LIN {X 0.037,Y -515.295,Z 622.606,A 0.000,B 0.000,C 90.000,E1 325.022} C_DIS
LIN {X 0.251,Y -517.921,Z 622.601,A 0.000,B 0.000,C 90.000,E1 324.116} C_DIS
LIN {X 0.091,Y -520.064,Z 622.598,A 0.000,B 0.000,C 90.000,E1 323.623} C_DIS
LIN {X 0.035,Y -521.634,Z 622.596,A 0.000,B 0.000,C 90.000,E1 323.336} C_DIS
LIN {X 0.167,Y -524.111,Z 622.594,A 0.000,B 0.000,C 90.000,E1 322.924} C_DIS
LIN {X 0.183,Y -527.814,Z 622.592,A 0.000,B 0.000,C 90.000,E1 322.477} C_DIS
LIN {X 0.246,Y -531.406,Z 622.590,A 0.000,B 0.000,C 90.000,E1 322.110} C_DIS
LIN {X -0.214,Y -538.842,Z 622.586,A 0.000,B 0.000,C 90.000,E1 321.537} C_DIS
LIN {X -0.001,Y -548.855,Z 622.582,A 0.000,B 0.000,C 90.000,E1 320.723} C_DIS
LIN {X -0.006,Y -561.804,Z 622.576,A 0.000,B 0.000,C 90.000,E1 319.666} C_DIS
LIN {X -0.280,Y -573.310,Z 622.571,A 0.000,B 0.000,C 90.000,E1 318.771} C_DIS
LIN {X 0.089,Y -581.806,Z 622.567,A 0.000,B 0.000,C 90.000,E1 318.038} C_DIS
LIN {X -0.035,Y -595.533,Z 622.560,A 0.000,B 0.000,C 90.000,E1 316.863} C_DIS
LIN {X 0.149,Y -600.581,Z 622.558,A 0.000,B 0.000,C 90.000,E1 316.377} C_DIS
LIN {X -0.381,Y -605.341,Z 622.555,A 0.000,B 0.000,C 90.000,E1 315.972} C_DIS
LIN {X 0.005,Y -609.117,Z 622.553,A 0.000,B 0.000,C 90.000,E1 315.567} C_DIS
LIN {X 0.270,Y -612.804,Z 622.551,A 0.000,B 0.000,C 90.000,E1 315.162} C_DIS
LIN {X 0.162,Y -620.880,Z 622.546,A 0.000,B 0.000,C 90.000,E1 314.271} C_DIS
LIN {X 0.244,Y -626.155,Z 622.543,A 0.000,B 0.000,C 90.000,E1 313.623} C_DIS
LIN {X -0.183,Y -633.203,Z 622.538,A 0.000,B 0.000,C 90.000,E1 312.771} C_DIS
LIN {X -0.232,Y -643.744,Z 622.530,A 0.000,B 0.000,C 90.000,E1 311.391} C_DIS
LIN {X 0.027,Y -650.113,Z 622.525,A 0.000,B 0.000,C 90.000,E1 310.496} C_DIS
LIN {X -0.084,Y -654.219,Z 622.522,A 0.000,B 0.000,C 90.000,E1 309.886} C_DIS
LIN {X -0.165,Y -657.973,Z 622.518,A 0.000,B 0.000,C 90.000,E1 309.277} C_DIS
LIN {X 0.262,Y -660.763,Z 622.515,A 0.000,B 0.000,C 90.000,E1 308.749} C_DIS
LIN {X -0.223,Y -663.342,Z 622.513,A 0.000,B 0.000,C 90.000,E1 308.302} C_DIS
LIN {X 0.327,Y -666.913,Z 622.509,A 0.000,B 0.000,C 90.000,E1 307.523} C_DIS
LIN {X -0.018,Y -670.263,Z 622.505,A 0.000,B 0.000,C 90.000,E1 306.824} C_DIS
LIN {X -0.058,Y -672.250,Z 622.502,A 0.000,B 0.000,C 90.000,E1 306.343} C_DIS
LIN {X 0.053,Y -674.129,Z 622.499,A 0.000,B 0.000,C 90.000,E1 305.851} C_DIS
LIN {X -0.088,Y -678.458,Z 622.493,A 0.000,B 0.000,C 90.000,E1 304.659} C_DIS
LIN {X 0.027,Y -682.444,Z 622.486,A 0.000,B 0.000,C 90.000,E1 303.452} C_DIS
LIN {X 0.220,Y -687.004,Z 622.478,A 0.000,B 0.000,C 90.000,E1 302.005} C_DIS
LIN {X -0.102,Y -690.569,Z 622.471,A 0.000,B 0.000,C 90.000,E1 300.846} C_DIS
LIN {X -0.131,Y -694.008,Z 622.465,A 0.000,B 0.000,C 90.000,E1 299.667} C_DIS
LIN {X 0.257,Y -696.610,Z 622.460,A 0.000,B 0.000,C 90.000,E1 298.693} C_DIS
LIN {X 0.066,Y -699.038,Z 622.454,A 0.000,B 0.000,C 90.000,E1 297.769} C_DIS
LIN {X -0.073,Y -700.684,Z 622.450,A 0.000,B 0.000,C 90.000,E1 297.078} C_DIS
LIN {X 0.124,Y -701.960,Z 622.447,A 0.000,B 0.000,C 90.000,E1 296.360} C_DIS
LIN {X 0.021,Y -702.388,Z 622.443,A 0.000,B 0.000,C 90.000,E1 295.668} C_DIS
LIN {X -0.055,Y -701.388,Z 622.440,A 0.000,B 0.000,C 90.000,E1 295.207} C_DIS
LIN {X 0.220,Y -700.776,Z 622.439,A 0.000,B 0.000,C 90.000,E1 294.951} C_DIS
LIN {X 0.063,Y -700.167,Z 622.438,A 0.000,B 0.000,C 90.000,E1 294.847} C_DIS
LIN {X -0.033,Y -696.435,Z 622.436,A 0.000,B 0.000,C 90.000,E1 294.387} C_DIS
LIN {X 0.097,Y -695.352,Z 622.435,A 0.000,B 0.000,C 90.000,E1 294.259} C_DIS
LIN {X -0.060,Y -693.693,Z 622.434,A 0.000,B 0.000,C 90.000,E1 294.155} C_DIS
LIN {X 0.051,Y -685.859,Z 622.432,A 0.000,B 0.000,C 90.000,E1 293.823} C_DIS
LIN {X -0.131,Y -683.986,Z 622.432,A 0.000,B 0.000,C 90.000,E1 293.770} C_DIS
LIN {X 0.041,Y -681.247,Z 622.432,A 0.000,B 0.000,C 90.000,E1 293.695} C_DIS
LIN {X 0.143,Y -673.456,Z 622.431,A 0.000,B 0.000,C 90.000,E1 293.567} C_DIS
LIN {X -0.172,Y -661.933,Z 622.430,A 0.000,B 0.000,C 90.000,E1 293.462} C_DIS
LIN {X -0.398,Y -651.490,Z 622.430,A 0.000,B 0.000,C 90.000,E1 293.334} C_DIS
LIN {X -0.145,Y -638.015,Z 622.428,A 0.000,B 0.000,C 90.000,E1 293.078} C_DIS
LIN {X 0.168,Y -628.722,Z 622.427,A 0.000,B 0.000,C 90.000,E1 292.845} C_DIS
LIN {X 0.104,Y -618.631,Z 622.426,A 0.000,B 0.000,C 90.000,E1 292.589} C_DIS
LIN {X 0.185,Y -598.220,Z 622.422,A 0.000,B 0.000,C 90.000,E1 291.972} C_DIS
LIN {X -0.273,Y -579.057,Z 622.419,A 0.000,B 0.000,C 90.000,E1 291.408} C_DIS
LIN {X -0.092,Y -570.115,Z 622.418,A 0.000,B 0.000,C 90.000,E1 291.153} C_DIS
LIN {X 0.255,Y -564.217,Z 622.416,A 0.000,B 0.000,C 90.000,E1 290.918} C_DIS
LIN {X -0.226,Y -559.393,Z 622.415,A 0.000,B 0.000,C 90.000,E1 290.737} C_DIS
LIN {X -0.220,Y -557.509,Z 622.414,A 0.000,B 0.000,C 90.000,E1 290.556} C_DIS
LIN {X -0.260,Y -557.482,Z 622.414,A 0.000,B 0.000,C 90.000,E1 290.556} C_DIS
LIN {X -0.181,Y -556.688,Z 622.413,A 0.000,B 0.000,C 90.000,E1 290.301} C_DIS
LIN {X -0.192,Y -556.434,Z 622.410,A 0.000,B 0.000,C 90.000,E1 289.885} C_DIS
LIN {X -0.146,Y -556.540,Z 622.403,A 0.000,B 0.000,C 90.000,E1 288.489} C_DIS
LIN {X 0.138,Y -556.461,Z 622.396,A 0.000,B 0.000,C 90.000,E1 287.347} C_DIS
LIN {X 0.287,Y -555.998,Z 622.387,A 0.000,B 0.000,C 90.000,E1 285.662} C_DIS
LIN {X 0.274,Y -555.606,Z 622.383,A 0.000,B 0.000,C 90.000,E1 284.828} C_DIS
LIN {X 0.094,Y -554.764,Z 622.373,A 0.000,B 0.000,C 90.000,E1 283.175} C_DIS
LIN {X -0.229,Y -553.949,Z 622.364,A 0.000,B 0.000,C 90.000,E1 281.535} C_DIS
LIN {X -0.251,Y -553.218,Z 622.356,A 0.000,B 0.000,C 90.000,E1 280.141} C_DIS
LIN {X -0.277,Y -552.643,Z 622.348,A 0.000,B 0.000,C 90.000,E1 278.746} C_DIS
LIN {X -0.280,Y -551.847,Z 622.339,A 0.000,B 0.000,C 90.000,E1 277.068} C_DIS
LIN {X -0.117,Y -550.855,Z 622.325,A 0.000,B 0.000,C 90.000,E1 274.531} C_DIS
LIN {X 0.216,Y -550.493,Z 622.317,A 0.000,B 0.000,C 90.000,E1 273.094} C_DIS
LIN {X 0.070,Y -549.983,Z 622.306,A 0.000,B 0.000,C 90.000,E1 271.146} C_DIS
LIN {X -0.203,Y -549.523,Z 622.299,A 0.000,B 0.000,C 90.000,E1 269.771} C_DIS
LIN {X 0.062,Y -548.936,Z 622.291,A 0.000,B 0.000,C 90.000,E1 268.339} C_DIS
LIN {X -0.145,Y -548.266,Z 622.281,A 0.000,B 0.000,C 90.000,E1 266.674} C_DIS
LIN {X 0.225,Y -547.221,Z 622.271,A 0.000,B 0.000,C 90.000,E1 264.666} C_DIS
LIN {X 0.002,Y -546.285,Z 622.263,A 0.000,B 0.000,C 90.000,E1 263.280} C_DIS
LIN {X 0.203,Y -545.569,Z 622.258,A 0.000,B 0.000,C 90.000,E1 262.413} C_DIS
LIN {X -0.137,Y -544.456,Z 622.252,A 0.000,B 0.000,C 90.000,E1 261.319} C_DIS
LIN {X -0.165,Y -542.341,Z 622.241,A 0.000,B 0.000,C 90.000,E1 259.342} C_DIS
LIN {X -0.141,Y -540.599,Z 622.230,A 0.000,B 0.000,C 90.000,E1 257.353} C_DIS
LIN {X -0.180,Y -539.406,Z 622.222,A 0.000,B 0.000,C 90.000,E1 255.936} C_DIS
LIN {X -0.241,Y -538.058,Z 622.214,A 0.000,B 0.000,C 90.000,E1 254.519} C_DIS
LIN {X 0.018,Y -536.201,Z 622.204,A 0.000,B 0.000,C 90.000,E1 252.779} C_DIS
LIN {X -0.270,Y -534.499,Z 622.195,A 0.000,B 0.000,C 90.000,E1 251.094} C_DIS
LIN {X 0.160,Y -533.507,Z 622.190,A 0.000,B 0.000,C 90.000,E1 250.188} C_DIS
LIN {X -0.227,Y -531.914,Z 622.184,A 0.000,B 0.000,C 90.000,E1 249.082} C_DIS
LIN {X -0.141,Y -530.154,Z 622.177,A 0.000,B 0.000,C 90.000,E1 247.922} C_DIS
LIN {X -0.069,Y -528.699,Z 622.172,A 0.000,B 0.000,C 90.000,E1 247.050} C_DIS
LIN {X -0.145,Y -526.109,Z 622.164,A 0.000,B 0.000,C 90.000,E1 245.613} C_DIS
LIN {X -0.209,Y -523.755,Z 622.158,A 0.000,B 0.000,C 90.000,E1 244.460} C_DIS
LIN {X -0.155,Y -520.585,Z 622.150,A 0.000,B 0.000,C 90.000,E1 242.999} C_DIS
LIN {X -0.054,Y -518.007,Z 622.143,A 0.000,B 0.000,C 90.000,E1 241.820} C_DIS
LIN {X 0.123,Y -514.673,Z 622.135,A 0.000,B 0.000,C 90.000,E1 240.333} C_DIS
LIN {X 0.130,Y -511.907,Z 622.129,A 0.000,B 0.000,C 90.000,E1 239.154} C_DIS
LIN {X 0.254,Y -508.317,Z 622.121,A 0.000,B 0.000,C 90.000,E1 237.661} C_DIS
LIN {X -0.002,Y -505.300,Z 622.114,A 0.000,B 0.000,C 90.000,E1 236.501} C_DIS
LIN {X -0.132,Y -501.371,Z 622.106,A 0.000,B 0.000,C 90.000,E1 235.022} C_DIS
LIN {X 0.202,Y -498.167,Z 622.099,A 0.000,B 0.000,C 90.000,E1 233.783} C_DIS
LIN {X -0.053,Y -492.758,Z 622.087,A 0.000,B 0.000,C 90.000,E1 231.698} C_DIS
LIN {X 0.017,Y -488.116,Z 622.077,A 0.000,B 0.000,C 90.000,E1 229.865} C_DIS
LIN {X 0.244,Y -483.519,Z 622.067,A 0.000,B 0.000,C 90.000,E1 228.000} C_DIS
LIN {X 0.250,Y -479.755,Z 622.058,A 0.000,B 0.000,C 90.000,E1 226.458} C_DIS
LIN {X -0.185,Y -473.716,Z 622.044,A 0.000,B 0.000,C 90.000,E1 224.028} C_DIS
LIN {X -0.115,Y -468.101,Z 622.031,A 0.000,B 0.000,C 90.000,E1 221.515} C_DIS
LIN {X -0.289,Y -464.046,Z 622.020,A 0.000,B 0.000,C 90.000,E1 219.644} C_DIS
LIN {X 0.191,Y -459.363,Z 622.008,A 0.000,B 0.000,C 90.000,E1 217.363} C_DIS
LIN {X -0.021,Y -454.922,Z 621.995,A 0.000,B 0.000,C 90.000,E1 215.152} C_DIS
LIN {X 0.045,Y -451.450,Z 621.985,A 0.000,B 0.000,C 90.000,E1 213.214} C_DIS
LIN {X 0.237,Y -447.254,Z 621.972,A 0.000,B 0.000,C 90.000,E1 210.924} C_DIS
LIN {X -0.130,Y -443.251,Z 621.959,A 0.000,B 0.000,C 90.000,E1 208.693} C_DIS
LIN {X -0.092,Y -440.312,Z 621.950,A 0.000,B 0.000,C 90.000,E1 207.052} C_DIS
LIN {X -0.100,Y -436.884,Z 621.939,A 0.000,B 0.000,C 90.000,E1 205.079} C_DIS
LIN {X -0.148,Y -432.811,Z 621.926,A 0.000,B 0.000,C 90.000,E1 202.770} C_DIS
LIN {X -0.068,Y -428.851,Z 621.914,A 0.000,B 0.000,C 90.000,E1 200.429} C_DIS
LIN {X -0.050,Y -425.502,Z 621.902,A 0.000,B 0.000,C 90.000,E1 198.417} C_DIS
LIN {X -0.018,Y -421.373,Z 621.887,A 0.000,B 0.000,C 90.000,E1 195.717} C_DIS
LIN {X 0.095,Y -418.912,Z 621.878,A 0.000,B 0.000,C 90.000,E1 194.008} C_DIS
LIN {X 0.162,Y -416.310,Z 621.869,A 0.000,B 0.000,C 90.000,E1 192.299} C_DIS
LIN {X 0.171,Y -412.757,Z 621.855,A 0.000,B 0.000,C 90.000,E1 189.905} C_DIS
LIN {X -0.086,Y -410.939,Z 621.848,A 0.000,B 0.000,C 90.000,E1 188.568} C_DIS
LIN {X -0.002,Y -408.521,Z 621.838,A 0.000,B 0.000,C 90.000,E1 186.834} C_DIS
LIN {X -0.037,Y -405.413,Z 621.825,A 0.000,B 0.000,C 90.000,E1 184.416} C_DIS
LIN {X 0.131,Y -401.928,Z 621.807,A 0.000,B 0.000,C 90.000,E1 181.260} C_DIS
LIN {X 0.000,Y -398.479,Z 621.784,A 0.000,B 0.000,C 90.000,E1 177.078} C_DIS
LIN {X 0.028,Y -397.138,Z 621.768,A 0.000,B 0.000,C 90.000,E1 174.261} C_DIS
LIN {X 0.101,Y -396.359,Z 621.753,A 0.000,B 0.000,C 90.000,E1 171.432} C_DIS
LIN {X -0.070,Y -396.094,Z 621.741,A 0.000,B 0.000,C 90.000,E1 169.342} C_DIS
LIN {X -0.126,Y -396.150,Z 621.727,A 0.000,B 0.000,C 90.000,E1 166.881} C_DIS
LIN {X -0.017,Y -396.373,Z 621.717,A 0.000,B 0.000,C 90.000,E1 165.102} C_DIS
LIN {X -0.194,Y -396.915,Z 621.702,A 0.000,B 0.000,C 90.000,E1 162.308} C_DIS
LIN {X 0.130,Y -397.572,Z 621.686,A 0.000,B 0.000,C 90.000,E1 159.444} C_DIS
LIN {X -0.040,Y -398.239,Z 621.674,A 0.000,B 0.000,C 90.000,E1 157.358} C_DIS
LIN {X 0.107,Y -398.957,Z 621.663,A 0.000,B 0.000,C 90.000,E1 155.229} C_DIS
LIN {X 0.078,Y -399.627,Z 621.651,A 0.000,B 0.000,C 90.000,E1 153.127} C_DIS
LIN {X 0.006,Y -400.238,Z 621.641,A 0.000,B 0.000,C 90.000,E1 151.385} C_DIS
LIN {X 0.020,Y -400.895,Z 621.629,A 0.000,B 0.000,C 90.000,E1 149.282} C_DIS
LIN {X 0.016,Y -401.385,Z 621.620,A 0.000,B 0.000,C 90.000,E1 147.533} C_DIS
LIN {X -0.208,Y -402.079,Z 621.608,A 0.000,B 0.000,C 90.000,E1 145.468} C_DIS
LIN {X -0.066,Y -402.968,Z 621.594,A 0.000,B 0.000,C 90.000,E1 143.004} C_DIS
LIN {X 0.135,Y -403.740,Z 621.583,A 0.000,B 0.000,C 90.000,E1 140.884} C_DIS
LIN {X -0.221,Y -404.196,Z 621.575,A 0.000,B 0.000,C 90.000,E1 139.542} C_DIS
LIN {X 0.094,Y -404.676,Z 621.565,A 0.000,B 0.000,C 90.000,E1 137.757} C_DIS
LIN {X -0.026,Y -405.195,Z 621.554,A 0.000,B 0.000,C 90.000,E1 135.688} C_DIS
LIN {X -0.157,Y -405.754,Z 621.542,A 0.000,B 0.000,C 90.000,E1 133.623} C_DIS
LIN {X 0.027,Y -406.393,Z 621.531,A 0.000,B 0.000,C 90.000,E1 131.515} C_DIS
LIN {X -0.022,Y -407.715,Z 621.515,A 0.000,B 0.000,C 90.000,E1 128.749} C_DIS
LIN {X -0.108,Y -407.999,Z 621.514,A 0.000,B 0.000,C 90.000,E1 128.588} C_DIS
LIN {X -0.157,Y -415.479,Z 621.500,A 0.000,B 0.000,C 90.000,E1 126.011} C_DIS
LIN {X 0.150,Y -416.832,Z 621.497,A 0.000,B 0.000,C 90.000,E1 125.391} C_DIS
LIN {X 0.112,Y -416.849,Z 621.497,A 0.000,B 0.000,C 90.000,E1 125.391} C_DIS
LIN {X 0.064,Y -419.608,Z 621.495,A 0.000,B 0.000,C 90.000,E1 125.152} C_DIS
LIN {X 0.049,Y -423.179,Z 621.494,A 0.000,B 0.000,C 90.000,E1 124.898} C_DIS
LIN {X -0.086,Y -434.535,Z 621.490,A 0.000,B 0.000,C 90.000,E1 124.278} C_DIS
LIN {X 0.274,Y -448.017,Z 621.486,A 0.000,B 0.000,C 90.000,E1 123.499} C_DIS
LIN {X -0.074,Y -459.616,Z 621.483,A 0.000,B 0.000,C 90.000,E1 122.880} C_DIS
LIN {X -0.055,Y -467.786,Z 621.480,A 0.000,B 0.000,C 90.000,E1 122.388} C_DIS
LIN {X 0.095,Y -477.463,Z 621.477,A 0.000,B 0.000,C 90.000,E1 121.750} C_DIS
LIN {X -0.113,Y -487.059,Z 621.473,A 0.000,B 0.000,C 90.000,E1 121.131} C_DIS
LIN {X 0.220,Y -493.119,Z 621.471,A 0.000,B 0.000,C 90.000,E1 120.669} C_DIS
LIN {X 0.137,Y -500.735,Z 621.468,A 0.000,B 0.000,C 90.000,E1 120.129} C_DIS
LIN {X 0.213,Y -508.268,Z 621.464,A 0.000,B 0.000,C 90.000,E1 119.539} C_DIS
LIN {X 0.157,Y -517.164,Z 621.460,A 0.000,B 0.000,C 90.000,E1 118.821} C_DIS
LIN {X -0.067,Y -524.305,Z 621.457,A 0.000,B 0.000,C 90.000,E1 118.231} C_DIS
LIN {X -0.130,Y -529.608,Z 621.454,A 0.000,B 0.000,C 90.000,E1 117.769} C_DIS
LIN {X 0.072,Y -533.562,Z 621.452,A 0.000,B 0.000,C 90.000,E1 117.385} C_DIS
LIN {X 0.073,Y -537.635,Z 621.450,A 0.000,B 0.000,C 90.000,E1 117.001} C_DIS
LIN {X -0.028,Y -541.452,Z 621.448,A 0.000,B 0.000,C 90.000,E1 116.616} C_DIS
LIN {X -0.065,Y -547.379,Z 621.444,A 0.000,B 0.000,C 90.000,E1 115.976} C_DIS
LIN {X 0.002,Y -551.874,Z 621.441,A 0.000,B 0.000,C 90.000,E1 115.412} C_DIS
LIN {X -0.066,Y -556.755,Z 621.437,A 0.000,B 0.000,C 90.000,E1 114.719} C_DIS
LIN {X -0.089,Y -561.008,Z 621.433,A 0.000,B 0.000,C 90.000,E1 114.027} C_DIS
LIN {X -0.078,Y -564.792,Z 621.430,A 0.000,B 0.000,C 90.000,E1 113.334} C_DIS
LIN {X 0.305,Y -569.312,Z 621.424,A 0.000,B 0.000,C 90.000,E1 112.333} C_DIS
LIN {X 0.171,Y -572.370,Z 621.420,A 0.000,B 0.000,C 90.000,E1 111.663} C_DIS
LIN {X -0.019,Y -575.771,Z 621.416,A 0.000,B 0.000,C 90.000,E1 110.865} C_DIS
LIN {X -0.178,Y -578.897,Z 621.411,A 0.000,B 0.000,C 90.000,E1 110.066} C_DIS
LIN {X 0.239,Y -581.728,Z 621.407,A 0.000,B 0.000,C 90.000,E1 109.214} C_DIS
LIN {X 0.134,Y -584.316,Z 621.402,A 0.000,B 0.000,C 90.000,E1 108.417} C_DIS
LIN {X -0.133,Y -586.641,Z 621.398,A 0.000,B 0.000,C 90.000,E1 107.638} C_DIS
LIN {X 0.037,Y -589.416,Z 621.392,A 0.000,B 0.000,C 90.000,E1 106.551} C_DIS
LIN {X -0.234,Y -592.766,Z 621.385,A 0.000,B 0.000,C 90.000,E1 105.245} C_DIS
LIN {X 0.121,Y -599.129,Z 621.371,A 0.000,B 0.000,C 90.000,E1 102.827} C_DIS
LIN {X -0.093,Y -604.115,Z 621.361,A 0.000,B 0.000,C 90.000,E1 101.007} C_DIS
LIN {X -0.112,Y -606.982,Z 621.355,A 0.000,B 0.000,C 90.000,E1 99.962} C_DIS
LIN {X -0.086,Y -609.693,Z 621.350,A 0.000,B 0.000,C 90.000,E1 98.916} C_DIS
LIN {X 0.232,Y -612.789,Z 621.342,A 0.000,B 0.000,C 90.000,E1 97.587} C_DIS
LIN {X 0.257,Y -615.216,Z 621.337,A 0.000,B 0.000,C 90.000,E1 96.549} C_DIS
LIN {X 0.054,Y -617.896,Z 621.329,A 0.000,B 0.000,C 90.000,E1 95.277} C_DIS
LIN {X -0.175,Y -620.149,Z 621.322,A 0.000,B 0.000,C 90.000,E1 94.012} C_DIS
LIN {X 0.210,Y -622.190,Z 621.315,A 0.000,B 0.000,C 90.000,E1 92.694} C_DIS
LIN {X -0.049,Y -623.264,Z 621.311,A 0.000,B 0.000,C 90.000,E1 91.949} C_DIS
LIN {X -0.231,Y -624.697,Z 621.304,A 0.000,B 0.000,C 90.000,E1 90.688} C_DIS
LIN {X 0.164,Y -625.371,Z 621.299,A 0.000,B 0.000,C 90.000,E1 89.885} C_DIS
LIN {X -0.061,Y -625.828,Z 621.295,A 0.000,B 0.000,C 90.000,E1 89.141} C_DIS
LIN {X 0.079,Y -626.134,Z 621.290,A 0.000,B 0.000,C 90.000,E1 88.108} C_DIS
LIN {X -0.141,Y -626.233,Z 621.285,A 0.000,B 0.000,C 90.000,E1 87.364} C_DIS
LIN {X -0.280,Y -625.978,Z 621.278,A 0.000,B 0.000,C 90.000,E1 86.102} C_DIS
LIN {X -0.091,Y -625.396,Z 621.273,A 0.000,B 0.000,C 90.000,E1 85.065} C_DIS
LIN {X -0.197,Y -624.514,Z 621.266,A 0.000,B 0.000,C 90.000,E1 83.799} C_DIS
LIN {X 0.207,Y -623.838,Z 621.261,A 0.000,B 0.000,C 90.000,E1 82.996} C_DIS
LIN {X -0.167,Y -622.716,Z 621.256,A 0.000,B 0.000,C 90.000,E1 82.008} C_DIS
LIN {X -0.093,Y -622.057,Z 621.253,A 0.000,B 0.000,C 90.000,E1 81.489} C_DIS
LIN {X -0.094,Y -620.032,Z 621.246,A 0.000,B 0.000,C 90.000,E1 80.208} C_DIS
LIN {X -0.123,Y -617.730,Z 621.238,A 0.000,B 0.000,C 90.000,E1 78.926} C_DIS
LIN {X 0.035,Y -615.748,Z 621.233,A 0.000,B 0.000,C 90.000,E1 77.881} C_DIS
LIN {X 0.044,Y -612.979,Z 621.226,A 0.000,B 0.000,C 90.000,E1 76.589} C_DIS
LIN {X -0.189,Y -610.552,Z 621.220,A 0.000,B 0.000,C 90.000,E1 75.574} C_DIS
LIN {X 0.239,Y -608.717,Z 621.215,A 0.000,B 0.000,C 90.000,E1 74.755} C_DIS
LIN {X -0.307,Y -605.438,Z 621.208,A 0.000,B 0.000,C 90.000,E1 73.504} C_DIS
LIN {X 0.217,Y -603.288,Z 621.204,A 0.000,B 0.000,C 90.000,E1 72.670} C_DIS
LIN {X 0.042,Y -600.097,Z 621.198,A 0.000,B 0.000,C 90.000,E1 71.638} C_DIS
LIN {X 0.227,Y -598.296,Z 621.195,A 0.000,B 0.000,C 90.000,E1 71.094} C_DIS
LIN {X -0.166,Y -596.467,Z 621.192,A 0.000,B 0.000,C 90.000,E1 70.604} C_DIS
LIN {X 0.131,Y -592.290,Z 621.186,A 0.000,B 0.000,C 90.000,E1 69.518} C_DIS
LIN {X -0.298,Y -590.123,Z 621.183,A 0.000,B 0.000,C 90.000,E1 69.028} C_DIS
LIN {X -0.095,Y -586.585,Z 621.179,A 0.000,B 0.000,C 90.000,E1 68.209} C_DIS
LIN {X 0.262,Y -581.568,Z 621.173,A 0.000,B 0.000,C 90.000,E1 67.102} C_DIS
LIN {X -0.312,Y -578.201,Z 621.169,A 0.000,B 0.000,C 90.000,E1 66.485} C_DIS
LIN {X -0.152,Y -574.584,Z 621.165,A 0.000,B 0.000,C 90.000,E1 65.793} C_DIS
LIN {X 0.062,Y -569.782,Z 621.161,A 0.000,B 0.000,C 90.000,E1 64.973} C_DIS
LIN {X 0.234,Y -566.232,Z 621.158,A 0.000,B 0.000,C 90.000,E1 64.409} C_DIS
LIN {X -0.226,Y -561.362,Z 621.154,A 0.000,B 0.000,C 90.000,E1 63.768} C_DIS
LIN {X -0.121,Y -557.133,Z 621.151,A 0.000,B 0.000,C 90.000,E1 63.204} C_DIS
LIN {X 0.202,Y -552.364,Z 621.148,A 0.000,B 0.000,C 90.000,E1 62.615} C_DIS
LIN {X 0.003,Y -548.633,Z 621.146,A 0.000,B 0.000,C 90.000,E1 62.231} C_DIS
LIN {X 0.168,Y -543.512,Z 621.143,A 0.000,B 0.000,C 90.000,E1 61.719} C_DIS
LIN {X 0.162,Y -537.977,Z 621.140,A 0.000,B 0.000,C 90.000,E1 61.257} C_DIS
LIN {X 0.115,Y -531.683,Z 621.138,A 0.000,B 0.000,C 90.000,E1 60.795} C_DIS
LIN {X 0.037,Y -524.887,Z 621.136,A 0.000,B 0.000,C 90.000,E1 60.383} C_DIS
LIN {X 0.104,Y -518.305,Z 621.133,A 0.000,B 0.000,C 90.000,E1 59.999} C_DIS
LIN {X -0.043,Y -513.243,Z 621.132,A 0.000,B 0.000,C 90.000,E1 59.744} C_DIS
LIN {X -0.144,Y -506.314,Z 621.130,A 0.000,B 0.000,C 90.000,E1 59.410} C_DIS
LIN {X 0.023,Y -486.255,Z 621.125,A 0.000,B 0.000,C 90.000,E1 58.408} C_DIS
LIN {X -0.053,Y -467.750,Z 621.119,A 0.000,B 0.000,C 90.000,E1 57.502} C_DIS
LIN {X -0.089,Y -454.702,Z 621.116,A 0.000,B 0.000,C 90.000,E1 56.834} C_DIS
LIN {X 0.053,Y -443.273,Z 621.112,A 0.000,B 0.000,C 90.000,E1 56.215} C_DIS
LIN {X 0.010,Y -443.243,Z 621.112,A 0.000,B 0.000,C 90.000,E1 56.215} C_DIS
LIN {X -0.219,Y -434.014,Z 621.090,A 0.000,B 0.000,C 90.000,E1 52.190} C_DIS
LIN {X 0.230,Y -431.546,Z 621.082,A 0.000,B 0.000,C 90.000,E1 50.803} C_DIS
LIN {X -0.063,Y -427.434,Z 621.073,A 0.000,B 0.000,C 90.000,E1 49.175} C_DIS
LIN {X -0.070,Y -428.168,Z 621.066,A 0.000,B 0.000,C 90.000,E1 47.796} C_DIS
LIN {X -0.240,Y -428.998,Z 621.054,A 0.000,B 0.000,C 90.000,E1 45.810} C_DIS
LIN {X 0.073,Y -430.004,Z 621.039,A 0.000,B 0.000,C 90.000,E1 43.095} C_DIS
LIN {X -0.095,Y -431.047,Z 621.027,A 0.000,B 0.000,C 90.000,E1 40.782} C_DIS
LIN {X -0.098,Y -431.845,Z 621.017,A 0.000,B 0.000,C 90.000,E1 39.116} C_DIS
LIN {X -0.027,Y -432.631,Z 621.008,A 0.000,B 0.000,C 90.000,E1 37.443} C_DIS
LIN {X -0.201,Y -433.303,Z 620.999,A 0.000,B 0.000,C 90.000,E1 35.804} C_DIS
LIN {X -0.025,Y -433.779,Z 620.991,A 0.000,B 0.000,C 90.000,E1 34.452} C_DIS
LIN {X 0.271,Y -434.223,Z 620.984,A 0.000,B 0.000,C 90.000,E1 33.086} C_DIS
LIN {X -0.005,Y -434.682,Z 620.975,A 0.000,B 0.000,C 90.000,E1 31.465} C_DIS
LIN {X -0.072,Y -435.413,Z 620.962,A 0.000,B 0.000,C 90.000,E1 29.155} C_DIS
LIN {X 0.237,Y -436.075,Z 620.951,A 0.000,B 0.000,C 90.000,E1 27.129} C_DIS
LIN {X -0.077,Y -436.556,Z 620.944,A 0.000,B 0.000,C 90.000,E1 25.848} C_DIS
LIN {X 0.250,Y -437.284,Z 620.933,A 0.000,B 0.000,C 90.000,E1 23.823} C_DIS
LIN {X 0.002,Y -437.954,Z 620.923,A 0.000,B 0.000,C 90.000,E1 22.206} C_DIS
LIN {X 0.015,Y -438.747,Z 620.914,A 0.000,B 0.000,C 90.000,E1 20.556} C_DIS
LIN {X 0.045,Y -439.483,Z 620.905,A 0.000,B 0.000,C 90.000,E1 18.906} C_DIS
LIN {X -0.089,Y -440.594,Z 620.892,A 0.000,B 0.000,C 90.000,E1 16.622} C_DIS
LIN {X 0.105,Y -441.926,Z 620.880,A 0.000,B 0.000,C 90.000,E1 14.300} C_DIS
LIN {X 0.012,Y -443.865,Z 620.863,A 0.000,B 0.000,C 90.000,E1 11.366} C_DIS
LIN {X -0.181,Y -446.236,Z 620.847,A 0.000,B 0.000,C 90.000,E1 8.454} C_DIS
LIN {X 0.084,Y -448.345,Z 620.834,A 0.000,B 0.000,C 90.000,E1 6.144} C_DIS
LIN {X -0.093,Y -450.622,Z 620.822,A 0.000,B 0.000,C 90.000,E1 3.898} C_DIS
LIN {X 0.171,Y -453.223,Z 620.809,A 0.000,B 0.000,C 90.000,E1 1.604} C_DIS
LIN {X -0.009,Y -457.314,Z 620.792,A 0.000,B 0.000,C 90.000,E1 358.511} C_DIS
LIN {X 0.188,Y -461.217,Z 620.778,A 0.000,B 0.000,C 90.000,E1 355.931} C_DIS
LIN {X 0.117,Y -464.371,Z 620.767,A 0.000,B 0.000,C 90.000,E1 354.033} C_DIS
LIN {X 0.170,Y -467.647,Z 620.756,A 0.000,B 0.000,C 90.000,E1 352.129} C_DIS
LIN {X 0.080,Y -470.240,Z 620.748,A 0.000,B 0.000,C 90.000,E1 350.566} C_DIS
LIN {X -0.056,Y -473.317,Z 620.737,A 0.000,B 0.000,C 90.000,E1 348.701} C_DIS
LIN {X -0.025,Y -476.570,Z 620.727,A 0.000,B 0.000,C 90.000,E1 346.825} C_DIS
LIN {X 0.192,Y -479.884,Z 620.716,A 0.000,B 0.000,C 90.000,E1 344.936} C_DIS
LIN {X 0.143,Y -483.949,Z 620.704,A 0.000,B 0.000,C 90.000,E1 342.779} C_DIS
LIN {X -0.118,Y -487.505,Z 620.694,A 0.000,B 0.000,C 90.000,E1 340.967} C_DIS
LIN {X -0.169,Y -490.500,Z 620.686,A 0.000,B 0.000,C 90.000,E1 339.444} C_DIS
LIN {X -0.212,Y -492.770,Z 620.679,A 0.000,B 0.000,C 90.000,E1 338.230} C_DIS
LIN {X 0.195,Y -495.429,Z 620.671,A 0.000,B 0.000,C 90.000,E1 336.666} C_DIS
LIN {X -0.054,Y -497.393,Z 620.664,A 0.000,B 0.000,C 90.000,E1 335.485} C_DIS
LIN {X -0.014,Y -499.705,Z 620.655,A 0.000,B 0.000,C 90.000,E1 333.973} C_DIS
LIN {X -0.161,Y -501.950,Z 620.647,A 0.000,B 0.000,C 90.000,E1 332.487} C_DIS
LIN {X -0.022,Y -504.136,Z 620.639,A 0.000,B 0.000,C 90.000,E1 330.973} C_DIS
LIN {X -0.002,Y -507.760,Z 620.625,A 0.000,B 0.000,C 90.000,E1 328.584} C_DIS
LIN {X 0.215,Y -513.566,Z 620.609,A 0.000,B 0.000,C 90.000,E1 325.595} C_DIS
LIN {X 0.036,Y -516.496,Z 620.602,A 0.000,B 0.000,C 90.000,E1 324.436} C_DIS
LIN {X 0.205,Y -518.373,Z 620.599,A 0.000,B 0.000,C 90.000,E1 323.829} C_DIS
LIN {X -0.056,Y -519.681,Z 620.597,A 0.000,B 0.000,C 90.000,E1 323.497} C_DIS
LIN {X 0.070,Y -520.340,Z 620.596,A 0.000,B 0.000,C 90.000,E1 323.336} C_DIS
LIN {X -0.264,Y -522.941,Z 620.594,A 0.000,B 0.000,C 90.000,E1 322.924} C_DIS
LIN {X -0.130,Y -523.540,Z 620.593,A 0.000,B 0.000,C 90.000,E1 322.763} C_DIS
LIN {X 0.005,Y -524.321,Z 620.592,A 0.000,B 0.000,C 90.000,E1 322.603} C_DIS
LIN {X 0.321,Y -527.429,Z 620.590,A 0.000,B 0.000,C 90.000,E1 322.190} C_DIS
LIN {X -0.212,Y -531.689,Z 620.588,A 0.000,B 0.000,C 90.000,E1 321.823} C_DIS
LIN {X 0.063,Y -537.429,Z 620.585,A 0.000,B 0.000,C 90.000,E1 321.295} C_DIS
LIN {X 0.004,Y -545.975,Z 620.581,A 0.000,B 0.000,C 90.000,E1 320.642} C_DIS
LIN {X 0.040,Y -558.958,Z 620.576,A 0.000,B 0.000,C 90.000,E1 319.585} C_DIS
LIN {X -0.165,Y -571.909,Z 620.570,A 0.000,B 0.000,C 90.000,E1 318.566} C_DIS
LIN {X -0.122,Y -581.805,Z 620.565,A 0.000,B 0.000,C 90.000,E1 317.757} C_DIS
LIN {X 0.080,Y -594.049,Z 620.560,A 0.000,B 0.000,C 90.000,E1 316.701} C_DIS
LIN {X 0.198,Y -601.966,Z 620.556,A 0.000,B 0.000,C 90.000,E1 315.972} C_DIS
LIN {X 0.160,Y -607.123,Z 620.553,A 0.000,B 0.000,C 90.000,E1 315.486} C_DIS
LIN {X -0.057,Y -612.012,Z 620.550,A 0.000,B 0.000,C 90.000,E1 315.000} C_DIS
LIN {X -0.038,Y -619.012,Z 620.546,A 0.000,B 0.000,C 90.000,E1 314.231} C_DIS
LIN {X 0.041,Y -624.472,Z 620.542,A 0.000,B 0.000,C 90.000,E1 313.581} C_DIS
LIN {X 0.031,Y -631.632,Z 620.537,A 0.000,B 0.000,C 90.000,E1 312.690} C_DIS
LIN {X 0.161,Y -640.319,Z 620.531,A 0.000,B 0.000,C 90.000,E1 311.553} C_DIS
LIN {X -0.026,Y -645.031,Z 620.528,A 0.000,B 0.000,C 90.000,E1 310.943} C_DIS
LIN {X 0.247,Y -650.462,Z 620.523,A 0.000,B 0.000,C 90.000,E1 310.172} C_DIS
LIN {X 0.136,Y -654.522,Z 620.520,A 0.000,B 0.000,C 90.000,E1 309.564} C_DIS
LIN {X 0.103,Y -656.809,Z 620.518,A 0.000,B 0.000,C 90.000,E1 309.197} C_DIS
LIN {X 0.110,Y -659.666,Z 620.515,A 0.000,B 0.000,C 90.000,E1 308.705} C_DIS
LIN {X 0.066,Y -662.922,Z 620.512,A 0.000,B 0.000,C 90.000,E1 308.096} C_DIS
LIN {X 0.089,Y -666.557,Z 620.508,A 0.000,B 0.000,C 90.000,E1 307.363} C_DIS
LIN {X 0.164,Y -668.876,Z 620.505,A 0.000,B 0.000,C 90.000,E1 306.870} C_DIS
LIN {X 0.256,Y -670.976,Z 620.502,A 0.000,B 0.000,C 90.000,E1 306.377} C_DIS
LIN {X -0.048,Y -673.784,Z 620.498,A 0.000,B 0.000,C 90.000,E1 305.678} C_DIS
LIN {X 0.218,Y -677.337,Z 620.493,A 0.000,B 0.000,C 90.000,E1 304.692} C_DIS
LIN {X 0.136,Y -681.412,Z 620.486,A 0.000,B 0.000,C 90.000,E1 303.499} C_DIS
LIN {X 0.114,Y -684.478,Z 620.481,A 0.000,B 0.000,C 90.000,E1 302.546} C_DIS
LIN {X 0.131,Y -687.507,Z 620.476,A 0.000,B 0.000,C 90.000,E1 301.592} C_DIS
LIN {X 0.056,Y -691.132,Z 620.469,A 0.000,B 0.000,C 90.000,E1 300.413} C_DIS
LIN {X 0.390,Y -694.586,Z 620.462,A 0.000,B 0.000,C 90.000,E1 299.205} C_DIS
LIN {X 0.102,Y -697.782,Z 620.456,A 0.000,B 0.000,C 90.000,E1 298.052} C_DIS
LIN {X -0.076,Y -700.147,Z 620.451,A 0.000,B 0.000,C 90.000,E1 297.129} C_DIS
LIN {X 0.113,Y -701.484,Z 620.447,A 0.000,B 0.000,C 90.000,E1 296.411} C_DIS
LIN {X 0.001,Y -702.009,Z 620.443,A 0.000,B 0.000,C 90.000,E1 295.720} C_DIS
LIN {X 0.278,Y -701.608,Z 620.442,A 0.000,B 0.000,C 90.000,E1 295.463} C_DIS
LIN {X -0.102,Y -700.509,Z 620.439,A 0.000,B 0.000,C 90.000,E1 295.027} C_DIS
LIN {X 0.035,Y -699.981,Z 620.438,A 0.000,B 0.000,C 90.000,E1 294.899} C_DIS
LIN {X -0.195,Y -697.305,Z 620.436,A 0.000,B 0.000,C 90.000,E1 294.567} C_DIS
LIN {X -0.221,Y -695.398,Z 620.435,A 0.000,B 0.000,C 90.000,E1 294.335} C_DIS
LIN {X -0.093,Y -693.956,Z 620.435,A 0.000,B 0.000,C 90.000,E1 294.207} C_DIS
LIN {X 0.035,Y -691.551,Z 620.434,A 0.000,B 0.000,C 90.000,E1 294.079} C_DIS
LIN {X 0.250,Y -684.445,Z 620.432,A 0.000,B 0.000,C 90.000,E1 293.770} C_DIS
LIN {X 0.071,Y -681.855,Z 620.432,A 0.000,B 0.000,C 90.000,E1 293.718} C_DIS
LIN {X 0.102,Y -674.043,Z 620.431,A 0.000,B 0.000,C 90.000,E1 293.590} C_DIS
LIN {X -0.051,Y -661.971,Z 620.430,A 0.000,B 0.000,C 90.000,E1 293.462} C_DIS
LIN {X -0.266,Y -651.534,Z 620.430,A 0.000,B 0.000,C 90.000,E1 293.334} C_DIS
LIN {X -0.020,Y -638.002,Z 620.428,A 0.000,B 0.000,C 90.000,E1 293.078} C_DIS
LIN {X -0.324,Y -628.579,Z 620.427,A 0.000,B 0.000,C 90.000,E1 292.898} C_DIS
LIN {X -0.040,Y -615.080,Z 620.425,A 0.000,B 0.000,C 90.000,E1 292.514} C_DIS
LIN {X -0.147,Y -580.817,Z 620.419,A 0.000,B 0.000,C 90.000,E1 291.461} C_DIS
LIN {X 0.069,Y -575.102,Z 620.418,A 0.000,B 0.000,C 90.000,E1 291.280} C_DIS
LIN {X -0.044,Y -569.926,Z 620.418,A 0.000,B 0.000,C 90.000,E1 291.153} C_DIS
LIN {X 0.337,Y -565.515,Z 620.417,A 0.000,B 0.000,C 90.000,E1 290.972} C_DIS
LIN {X -0.133,Y -559.483,Z 620.415,A 0.000,B 0.000,C 90.000,E1 290.737} C_DIS
LIN {X -0.197,Y -557.563,Z 620.414,A 0.000,B 0.000,C 90.000,E1 290.556} C_DIS
LIN {X -0.237,Y -557.523,Z 620.414,A 0.000,B 0.000,C 90.000,E1 290.556} C_DIS
LIN {X 0.012,Y -556.821,Z 620.413,A 0.000,B 0.000,C 90.000,E1 290.301} C_DIS
LIN {X 0.003,Y -556.610,Z 620.411,A 0.000,B 0.000,C 90.000,E1 289.885} C_DIS
LIN {X 0.051,Y -556.688,Z 620.403,A 0.000,B 0.000,C 90.000,E1 288.489} C_DIS
LIN {X -0.193,Y -556.613,Z 620.397,A 0.000,B 0.000,C 90.000,E1 287.402} C_DIS
LIN {X 0.212,Y -556.233,Z 620.389,A 0.000,B 0.000,C 90.000,E1 285.969} C_DIS
LIN {X -0.201,Y -555.741,Z 620.383,A 0.000,B 0.000,C 90.000,E1 284.898} C_DIS
LIN {X 0.044,Y -555.072,Z 620.375,A 0.000,B 0.000,C 90.000,E1 283.480} C_DIS
LIN {X -0.146,Y -554.216,Z 620.366,A 0.000,B 0.000,C 90.000,E1 281.827} C_DIS
LIN {X -0.063,Y -553.504,Z 620.358,A 0.000,B 0.000,C 90.000,E1 280.423} C_DIS
LIN {X -0.063,Y -552.750,Z 620.349,A 0.000,B 0.000,C 90.000,E1 278.746} C_DIS
LIN {X 0.047,Y -551.820,Z 620.338,A 0.000,B 0.000,C 90.000,E1 276.777} C_DIS
LIN {X 0.005,Y -551.051,Z 620.327,A 0.000,B 0.000,C 90.000,E1 274.821} C_DIS
LIN {X -0.143,Y -550.592,Z 620.318,A 0.000,B 0.000,C 90.000,E1 273.154} C_DIS
LIN {X -0.257,Y -550.084,Z 620.307,A 0.000,B 0.000,C 90.000,E1 271.203} C_DIS
LIN {X 0.021,Y -549.627,Z 620.299,A 0.000,B 0.000,C 90.000,E1 269.771} C_DIS
LIN {X -0.260,Y -549.040,Z 620.291,A 0.000,B 0.000,C 90.000,E1 268.396} C_DIS
LIN {X 0.084,Y -548.372,Z 620.282,A 0.000,B 0.000,C 90.000,E1 266.674} C_DIS
LIN {X -0.127,Y -547.505,Z 620.272,A 0.000,B 0.000,C 90.000,E1 265.008} C_DIS
LIN {X 0.145,Y -546.617,Z 620.264,A 0.000,B 0.000,C 90.000,E1 263.571} C_DIS
LIN {X -0.194,Y -545.992,Z 620.260,A 0.000,B 0.000,C 90.000,E1 262.761} C_DIS
LIN {X 0.100,Y -544.607,Z 620.252,A 0.000,B 0.000,C 90.000,E1 261.319} C_DIS
LIN {X -0.010,Y -542.805,Z 620.242,A 0.000,B 0.000,C 90.000,E1 259.634} C_DIS
LIN {X 0.102,Y -540.772,Z 620.230,A 0.000,B 0.000,C 90.000,E1 257.353} C_DIS
LIN {X 0.065,Y -539.549,Z 620.222,A 0.000,B 0.000,C 90.000,E1 255.936} C_DIS
LIN {X 0.006,Y -538.204,Z 620.214,A 0.000,B 0.000,C 90.000,E1 254.519} C_DIS
LIN {X 0.266,Y -536.345,Z 620.205,A 0.000,B 0.000,C 90.000,E1 252.779} C_DIS
LIN {X -0.019,Y -534.644,Z 620.195,A 0.000,B 0.000,C 90.000,E1 251.094} C_DIS
LIN {X -0.090,Y -533.656,Z 620.190,A 0.000,B 0.000,C 90.000,E1 250.242} C_DIS
LIN {X -0.171,Y -532.460,Z 620.185,A 0.000,B 0.000,C 90.000,E1 249.390} C_DIS
LIN {X -0.076,Y -530.740,Z 620.179,A 0.000,B 0.000,C 90.000,E1 248.230} C_DIS
LIN {X 0.187,Y -528.803,Z 620.173,A 0.000,B 0.000,C 90.000,E1 247.050} C_DIS
LIN {X 0.112,Y -526.218,Z 620.165,A 0.000,B 0.000,C 90.000,E1 245.613} C_DIS
LIN {X 0.047,Y -523.847,Z 620.158,A 0.000,B 0.000,C 90.000,E1 244.460} C_DIS
LIN {X -0.043,Y -521.325,Z 620.152,A 0.000,B 0.000,C 90.000,E1 243.307} C_DIS
LIN {X -0.170,Y -518.766,Z 620.145,A 0.000,B 0.000,C 90.000,E1 242.153} C_DIS
LIN {X 0.020,Y -515.447,Z 620.137,A 0.000,B 0.000,C 90.000,E1 240.667} C_DIS
LIN {X 0.039,Y -512.692,Z 620.131,A 0.000,B 0.000,C 90.000,E1 239.488} C_DIS
LIN {X -0.160,Y -509.864,Z 620.124,A 0.000,B 0.000,C 90.000,E1 238.329} C_DIS
LIN {X -0.065,Y -506.149,Z 620.116,A 0.000,B 0.000,C 90.000,E1 236.834} C_DIS
LIN {X 0.237,Y -502.211,Z 620.107,A 0.000,B 0.000,C 90.000,E1 235.308} C_DIS
LIN {X 0.176,Y -499.011,Z 620.101,A 0.000,B 0.000,C 90.000,E1 234.116} C_DIS
LIN {X 0.052,Y -491.991,Z 620.086,A 0.000,B 0.000,C 90.000,E1 231.412} C_DIS
LIN {X -0.106,Y -488.119,Z 620.077,A 0.000,B 0.000,C 90.000,E1 229.908} C_DIS
LIN {X -0.191,Y -483.513,Z 620.067,A 0.000,B 0.000,C 90.000,E1 228.081} C_DIS
LIN {X -0.183,Y -479.741,Z 620.058,A 0.000,B 0.000,C 90.000,E1 226.539} C_DIS
LIN {X 0.057,Y -473.711,Z 620.045,A 0.000,B 0.000,C 90.000,E1 224.028} C_DIS
LIN {X 0.048,Y -468.768,Z 620.033,A 0.000,B 0.000,C 90.000,E1 221.838} C_DIS
LIN {X 0.133,Y -465.348,Z 620.024,A 0.000,B 0.000,C 90.000,E1 220.253} C_DIS
LIN {X 0.148,Y -461.915,Z 620.015,A 0.000,B 0.000,C 90.000,E1 218.669} C_DIS
LIN {X 0.164,Y -458.675,Z 620.006,A 0.000,B 0.000,C 90.000,E1 217.076} C_DIS
LIN {X -0.067,Y -454.263,Z 619.994,A 0.000,B 0.000,C 90.000,E1 214.865} C_DIS
LIN {X 0.023,Y -451.388,Z 619.985,A 0.000,B 0.000,C 90.000,E1 213.245} C_DIS
LIN {X -0.154,Y -447.191,Z 619.972,A 0.000,B 0.000,C 90.000,E1 211.003} C_DIS
LIN {X 0.089,Y -443.192,Z 619.960,A 0.000,B 0.000,C 90.000,E1 208.693} C_DIS
LIN {X 0.082,Y -440.860,Z 619.952,A 0.000,B 0.000,C 90.000,E1 207.385} C_DIS
LIN {X 0.093,Y -437.399,Z 619.941,A 0.000,B 0.000,C 90.000,E1 205.412} C_DIS
LIN {X 0.062,Y -432.750,Z 619.927,A 0.000,B 0.000,C 90.000,E1 202.770} C_DIS
LIN {X 0.138,Y -428.825,Z 619.914,A 0.000,B 0.000,C 90.000,E1 200.429} C_DIS
LIN {X -0.053,Y -424.938,Z 619.901,A 0.000,B 0.000,C 90.000,E1 198.109} C_DIS
LIN {X 0.008,Y -421.852,Z 619.889,A 0.000,B 0.000,C 90.000,E1 196.079} C_DIS
LIN {X 0.237,Y -419.439,Z 619.880,A 0.000,B 0.000,C 90.000,E1 194.356} C_DIS
LIN {X -0.097,Y -416.866,Z 619.871,A 0.000,B 0.000,C 90.000,E1 192.703} C_DIS
LIN {X -0.079,Y -413.295,Z 619.857,A 0.000,B 0.000,C 90.000,E1 190.310} C_DIS
LIN {X 0.113,Y -410.978,Z 619.848,A 0.000,B 0.000,C 90.000,E1 188.568} C_DIS
LIN {X 0.197,Y -408.586,Z 619.838,A 0.000,B 0.000,C 90.000,E1 186.834} C_DIS
LIN {X 0.162,Y -405.481,Z 619.825,A 0.000,B 0.000,C 90.000,E1 184.416} C_DIS
LIN {X -0.071,Y -402.010,Z 619.807,A 0.000,B 0.000,C 90.000,E1 181.318} C_DIS
LIN {X -0.196,Y -398.594,Z 619.784,A 0.000,B 0.000,C 90.000,E1 177.135} C_DIS
LIN {X 0.133,Y -397.002,Z 619.764,A 0.000,B 0.000,C 90.000,E1 173.571} C_DIS
LIN {X -0.165,Y -396.317,Z 619.747,A 0.000,B 0.000,C 90.000,E1 170.443} C_DIS
LIN {X 0.086,Y -396.251,Z 619.727,A 0.000,B 0.000,C 90.000,E1 166.881} C_DIS
LIN {X 0.158,Y -396.530,Z 619.715,A 0.000,B 0.000,C 90.000,E1 164.755} C_DIS
LIN {X 0.025,Y -397.056,Z 619.702,A 0.000,B 0.000,C 90.000,E1 162.308} C_DIS
LIN {X 0.144,Y -397.616,Z 619.688,A 0.000,B 0.000,C 90.000,E1 159.826} C_DIS
LIN {X 0.117,Y -398.287,Z 619.676,A 0.000,B 0.000,C 90.000,E1 157.720} C_DIS
LIN {X 0.109,Y -398.996,Z 619.665,A 0.000,B 0.000,C 90.000,E1 155.613} C_DIS
LIN {X 0.080,Y -399.734,Z 619.653,A 0.000,B 0.000,C 90.000,E1 153.512} C_DIS
LIN {X -0.105,Y -400.453,Z 619.641,A 0.000,B 0.000,C 90.000,E1 151.435} C_DIS
LIN {X -0.077,Y -401.105,Z 619.630,A 0.000,B 0.000,C 90.000,E1 149.331} C_DIS
LIN {X -0.181,Y -401.702,Z 619.618,A 0.000,B 0.000,C 90.000,E1 147.248} C_DIS
LIN {X 0.050,Y -402.280,Z 619.608,A 0.000,B 0.000,C 90.000,E1 145.468} C_DIS
LIN {X -0.124,Y -403.159,Z 619.595,A 0.000,B 0.000,C 90.000,E1 143.050} C_DIS
LIN {X 0.091,Y -403.903,Z 619.583,A 0.000,B 0.000,C 90.000,E1 140.928} C_DIS
LIN {X -0.125,Y -404.508,Z 619.573,A 0.000,B 0.000,C 90.000,E1 139.218} C_DIS
LIN {X -0.071,Y -404.909,Z 619.564,A 0.000,B 0.000,C 90.000,E1 137.472} C_DIS
LIN {X -0.201,Y -405.413,Z 619.552,A 0.000,B 0.000,C 90.000,E1 135.405} C_DIS
LIN {X -0.037,Y -405.967,Z 619.541,A 0.000,B 0.000,C 90.000,E1 133.299} C_DIS
LIN {X 0.044,Y -406.476,Z 619.531,A 0.000,B 0.000,C 90.000,E1 131.553} C_DIS
LIN {X 0.010,Y -407.659,Z 619.516,A 0.000,B 0.000,C 90.000,E1 128.785} C_DIS
LIN {X -0.075,Y -407.889,Z 619.515,A 0.000,B 0.000,C 90.000,E1 128.624} C_DIS
LIN {X 0.133,Y -415.355,Z 619.500,A 0.000,B 0.000,C 90.000,E1 126.011} C_DIS
LIN {X 0.080,Y -417.522,Z 619.495,A 0.000,B 0.000,C 90.000,E1 125.105} C_DIS
LIN {X 0.041,Y -417.543,Z 619.495,A 0.000,B 0.000,C 90.000,E1 125.105} C_DIS
LIN {X -0.155,Y -418.709,Z 619.495,A 0.000,B 0.000,C 90.000,E1 125.025} C_DIS
LIN {X 0.236,Y -423.787,Z 619.492,A 0.000,B 0.000,C 90.000,E1 124.612} C_DIS
LIN {X -0.265,Y -443.768,Z 619.486,A 0.000,B 0.000,C 90.000,E1 123.579} C_DIS
LIN {X -0.093,Y -453.257,Z 619.484,A 0.000,B 0.000,C 90.000,E1 123.038} C_DIS
LIN {X -0.050,Y -463.185,Z 619.480,A 0.000,B 0.000,C 90.000,E1 122.467} C_DIS
LIN {X 0.061,Y -471.311,Z 619.478,A 0.000,B 0.000,C 90.000,E1 121.957} C_DIS
LIN {X -0.148,Y -479.402,Z 619.475,A 0.000,B 0.000,C 90.000,E1 121.465} C_DIS
LIN {X -0.031,Y -488.476,Z 619.471,A 0.000,B 0.000,C 90.000,E1 120.846} C_DIS
LIN {X -0.010,Y -497.530,Z 619.468,A 0.000,B 0.000,C 90.000,E1 120.207} C_DIS
LIN {X -0.055,Y -502.113,Z 619.466,A 0.000,B 0.000,C 90.000,E1 119.873} C_DIS
LIN {X 0.230,Y -507.773,Z 619.464,A 0.000,B 0.000,C 90.000,E1 119.411} C_DIS
LIN {X -0.152,Y -516.628,Z 619.460,A 0.000,B 0.000,C 90.000,E1 118.743} C_DIS
LIN {X 0.033,Y -526.417,Z 619.455,A 0.000,B 0.000,C 90.000,E1 117.897} C_DIS
LIN {X -0.115,Y -533.097,Z 619.452,A 0.000,B 0.000,C 90.000,E1 117.308} C_DIS
LIN {X -0.104,Y -537.205,Z 619.450,A 0.000,B 0.000,C 90.000,E1 116.924} C_DIS
LIN {X 0.250,Y -542.401,Z 619.447,A 0.000,B 0.000,C 90.000,E1 116.360} C_DIS
LIN {X -0.007,Y -546.346,Z 619.444,A 0.000,B 0.000,C 90.000,E1 115.976} C_DIS
LIN {X 0.053,Y -551.050,Z 619.441,A 0.000,B 0.000,C 90.000,E1 115.412} C_DIS
LIN {X -0.022,Y -556.168,Z 619.437,A 0.000,B 0.000,C 90.000,E1 114.719} C_DIS
LIN {X -0.050,Y -560.559,Z 619.433,A 0.000,B 0.000,C 90.000,E1 114.027} C_DIS
LIN {X -0.042,Y -564.414,Z 619.430,A 0.000,B 0.000,C 90.000,E1 113.334} C_DIS
LIN {X -0.190,Y -569.078,Z 619.424,A 0.000,B 0.000,C 90.000,E1 112.386} C_DIS
LIN {X 0.027,Y -573.413,Z 619.419,A 0.000,B 0.000,C 90.000,E1 111.408} C_DIS
LIN {X 0.012,Y -575.687,Z 619.416,A 0.000,B 0.000,C 90.000,E1 110.865} C_DIS
LIN {X -0.149,Y -578.872,Z 619.411,A 0.000,B 0.000,C 90.000,E1 110.066} C_DIS
LIN {X -0.281,Y -581.774,Z 619.407,A 0.000,B 0.000,C 90.000,E1 109.268} C_DIS
LIN {X 0.165,Y -584.431,Z 619.402,A 0.000,B 0.000,C 90.000,E1 108.417} C_DIS
LIN {X 0.131,Y -587.574,Z 619.396,A 0.000,B 0.000,C 90.000,E1 107.347} C_DIS
LIN {X 0.006,Y -591.054,Z 619.389,A 0.000,B 0.000,C 90.000,E1 106.024} C_DIS
LIN {X -0.125,Y -598.735,Z 619.373,A 0.000,B 0.000,C 90.000,E1 103.119} C_DIS
LIN {X -0.098,Y -601.638,Z 619.367,A 0.000,B 0.000,C 90.000,E1 102.063} C_DIS
LIN {X -0.102,Y -606.025,Z 619.358,A 0.000,B 0.000,C 90.000,E1 100.489} C_DIS
LIN {X -0.085,Y -608.840,Z 619.352,A 0.000,B 0.000,C 90.000,E1 99.443} C_DIS
LIN {X 0.323,Y -610.841,Z 619.348,A 0.000,B 0.000,C 90.000,E1 98.624} C_DIS
LIN {X 0.052,Y -613.962,Z 619.341,A 0.000,B 0.000,C 90.000,E1 97.352} C_DIS
LIN {X 0.087,Y -616.363,Z 619.335,A 0.000,B 0.000,C 90.000,E1 96.315} C_DIS
LIN {X 0.154,Y -618.555,Z 619.329,A 0.000,B 0.000,C 90.000,E1 95.277} C_DIS
LIN {X -0.064,Y -620.842,Z 619.322,A 0.000,B 0.000,C 90.000,E1 94.012} C_DIS
LIN {X -0.288,Y -622.886,Z 619.315,A 0.000,B 0.000,C 90.000,E1 92.751} C_DIS
LIN {X 0.081,Y -623.963,Z 619.311,A 0.000,B 0.000,C 90.000,E1 91.949} C_DIS
LIN {X -0.088,Y -625.434,Z 619.304,A 0.000,B 0.000,C 90.000,E1 90.688} C_DIS
LIN {X -0.312,Y -626.112,Z 619.300,A 0.000,B 0.000,C 90.000,E1 89.943} C_DIS
LIN {X 0.098,Y -626.572,Z 619.295,A 0.000,B 0.000,C 90.000,E1 89.141} C_DIS
LIN {X 0.248,Y -626.852,Z 619.290,A 0.000,B 0.000,C 90.000,E1 88.108} C_DIS
LIN {X 0.034,Y -626.969,Z 619.285,A 0.000,B 0.000,C 90.000,E1 87.364} C_DIS
LIN {X -0.094,Y -626.704,Z 619.278,A 0.000,B 0.000,C 90.000,E1 86.102} C_DIS
LIN {X -0.185,Y -625.915,Z 619.271,A 0.000,B 0.000,C 90.000,E1 84.837} C_DIS
LIN {X -0.288,Y -624.966,Z 619.264,A 0.000,B 0.000,C 90.000,E1 83.571} C_DIS
LIN {X 0.195,Y -624.244,Z 619.260,A 0.000,B 0.000,C 90.000,E1 82.761} C_DIS
LIN {X 0.135,Y -622.664,Z 619.253,A 0.000,B 0.000,C 90.000,E1 81.489} C_DIS
LIN {X 0.143,Y -620.609,Z 619.246,A 0.000,B 0.000,C 90.000,E1 80.208} C_DIS
LIN {X -0.032,Y -619.218,Z 619.241,A 0.000,B 0.000,C 90.000,E1 79.454} C_DIS
LIN {X -0.085,Y -616.724,Z 619.234,A 0.000,B 0.000,C 90.000,E1 78.173} C_DIS
LIN {X 0.052,Y -615.644,Z 619.231,A 0.000,B 0.000,C 90.000,E1 77.645} C_DIS
LIN {X -0.295,Y -613.440,Z 619.226,A 0.000,B 0.000,C 90.000,E1 76.645} C_DIS
LIN {X -0.078,Y -610.957,Z 619.220,A 0.000,B 0.000,C 90.000,E1 75.589} C_DIS
LIN {X -0.082,Y -609.115,Z 619.216,A 0.000,B 0.000,C 90.000,E1 74.810} C_DIS
LIN {X -0.036,Y -605.752,Z 619.208,A 0.000,B 0.000,C 90.000,E1 73.504} C_DIS
LIN {X -0.086,Y -603.556,Z 619.204,A 0.000,B 0.000,C 90.000,E1 72.725} C_DIS
LIN {X 0.318,Y -600.277,Z 619.198,A 0.000,B 0.000,C 90.000,E1 71.638} C_DIS
LIN {X 0.032,Y -599.426,Z 619.197,A 0.000,B 0.000,C 90.000,E1 71.402} C_DIS
LIN {X 0.110,Y -596.570,Z 619.192,A 0.000,B 0.000,C 90.000,E1 70.604} C_DIS
LIN {X -0.041,Y -593.405,Z 619.188,A 0.000,B 0.000,C 90.000,E1 69.826} C_DIS
LIN {X -0.024,Y -590.092,Z 619.184,A 0.000,B 0.000,C 90.000,E1 69.028} C_DIS
LIN {X -0.101,Y -585.905,Z 619.178,A 0.000,B 0.000,C 90.000,E1 68.103} C_DIS
LIN {X 0.058,Y -582.065,Z 619.174,A 0.000,B 0.000,C 90.000,E1 67.283} C_DIS
LIN {X -0.050,Y -577.919,Z 619.169,A 0.000,B 0.000,C 90.000,E1 66.485} C_DIS
LIN {X 0.106,Y -574.199,Z 619.166,A 0.000,B 0.000,C 90.000,E1 65.793} C_DIS
LIN {X 0.226,Y -570.088,Z 619.162,A 0.000,B 0.000,C 90.000,E1 65.101} C_DIS
LIN {X -0.095,Y -565.553,Z 619.158,A 0.000,B 0.000,C 90.000,E1 64.460} C_DIS
LIN {X -0.051,Y -560.537,Z 619.154,A 0.000,B 0.000,C 90.000,E1 63.768} C_DIS
LIN {X 0.151,Y -557.366,Z 619.152,A 0.000,B 0.000,C 90.000,E1 63.332} C_DIS
LIN {X -0.019,Y -552.541,Z 619.149,A 0.000,B 0.000,C 90.000,E1 62.794} C_DIS
LIN {X 0.156,Y -547.280,Z 619.146,A 0.000,B 0.000,C 90.000,E1 62.231} C_DIS
LIN {X -0.015,Y -542.911,Z 619.144,A 0.000,B 0.000,C 90.000,E1 61.847} C_DIS
LIN {X 0.221,Y -535.840,Z 619.141,A 0.000,B 0.000,C 90.000,E1 61.257} C_DIS
LIN {X 0.127,Y -530.984,Z 619.139,A 0.000,B 0.000,C 90.000,E1 60.923} C_DIS
LIN {X -0.048,Y -524.333,Z 619.136,A 0.000,B 0.000,C 90.000,E1 60.539} C_DIS
LIN {X 0.270,Y -517.649,Z 619.134,A 0.000,B 0.000,C 90.000,E1 60.127} C_DIS
LIN {X -0.234,Y -509.128,Z 619.132,A 0.000,B 0.000,C 90.000,E1 59.744} C_DIS
LIN {X -0.003,Y -490.520,Z 619.127,A 0.000,B 0.000,C 90.000,E1 58.820} C_DIS
LIN {X -0.117,Y -478.593,Z 619.124,A 0.000,B 0.000,C 90.000,E1 58.250} C_DIS
LIN {X 0.114,Y -453.763,Z 619.117,A 0.000,B 0.000,C 90.000,E1 56.962} C_DIS
LIN {X -0.279,Y -443.906,Z 619.114,A 0.000,B 0.000,C 90.000,E1 56.501} C_DIS
LIN {X 0.294,Y -443.871,Z 619.114,A 0.000,B 0.000,C 90.000,E1 56.421} C_DIS
LIN {X 0.112,Y -434.507,Z 619.091,A 0.000,B 0.000,C 90.000,E1 52.396} C_DIS
LIN {X 0.223,Y -431.367,Z 619.082,A 0.000,B 0.000,C 90.000,E1 50.723} C_DIS
LIN {X -0.010,Y -427.835,Z 619.074,A 0.000,B 0.000,C 90.000,E1 49.337} C_DIS
LIN {X -0.009,Y -428.561,Z 619.067,A 0.000,B 0.000,C 90.000,E1 48.081} C_DIS
LIN {X 0.147,Y -429.434,Z 619.056,A 0.000,B 0.000,C 90.000,E1 46.053} C_DIS
LIN {X 0.236,Y -430.333,Z 619.043,A 0.000,B 0.000,C 90.000,E1 43.704} C_DIS
LIN {X -0.031,Y -430.949,Z 619.036,A 0.000,B 0.000,C 90.000,E1 42.405} C_DIS
LIN {X 0.180,Y -431.897,Z 619.024,A 0.000,B 0.000,C 90.000,E1 40.378} C_DIS
LIN {X -0.086,Y -432.699,Z 619.015,A 0.000,B 0.000,C 90.000,E1 38.749} C_DIS
LIN {X 0.084,Y -433.294,Z 619.008,A 0.000,B 0.000,C 90.000,E1 37.397} C_DIS
LIN {X 0.183,Y -433.975,Z 618.999,A 0.000,B 0.000,C 90.000,E1 35.724} C_DIS
LIN {X 0.123,Y -434.446,Z 618.991,A 0.000,B 0.000,C 90.000,E1 34.405} C_DIS
LIN {X 0.089,Y -434.917,Z 618.982,A 0.000,B 0.000,C 90.000,E1 32.752} C_DIS
LIN {X -0.125,Y -435.557,Z 618.969,A 0.000,B 0.000,C 90.000,E1 30.463} C_DIS
LIN {X -0.220,Y -436.049,Z 618.960,A 0.000,B 0.000,C 90.000,E1 28.821} C_DIS
LIN {X 0.098,Y -436.733,Z 618.949,A 0.000,B 0.000,C 90.000,E1 26.796} C_DIS
LIN {X 0.096,Y -437.646,Z 618.934,A 0.000,B 0.000,C 90.000,E1 24.155} C_DIS
LIN {X -0.130,Y -438.382,Z 618.923,A 0.000,B 0.000,C 90.000,E1 22.206} C_DIS
LIN {X -0.268,Y -439.271,Z 618.912,A 0.000,B 0.000,C 90.000,E1 20.248} C_DIS
LIN {X 0.186,Y -439.991,Z 618.903,A 0.000,B 0.000,C 90.000,E1 18.544} C_DIS
LIN {X -0.197,Y -440.931,Z 618.892,A 0.000,B 0.000,C 90.000,E1 16.622} C_DIS
LIN {X -0.144,Y -442.060,Z 618.881,A 0.000,B 0.000,C 90.000,E1 14.647} C_DIS
LIN {X 0.191,Y -443.925,Z 618.865,A 0.000,B 0.000,C 90.000,E1 11.658} C_DIS
LIN {X 0.004,Y -446.207,Z 618.849,A 0.000,B 0.000,C 90.000,E1 8.746} C_DIS
LIN {X -0.120,Y -448.273,Z 618.836,A 0.000,B 0.000,C 90.000,E1 6.486} C_DIS
LIN {X -0.159,Y -450.825,Z 618.822,A 0.000,B 0.000,C 90.000,E1 3.898} C_DIS
LIN {X 0.111,Y -453.396,Z 618.809,A 0.000,B 0.000,C 90.000,E1 1.604} C_DIS
LIN {X -0.192,Y -457.000,Z 618.794,A 0.000,B 0.000,C 90.000,E1 358.854} C_DIS
LIN {X -0.002,Y -460.833,Z 618.779,A 0.000,B 0.000,C 90.000,E1 356.274} C_DIS
LIN {X -0.084,Y -465.034,Z 618.765,A 0.000,B 0.000,C 90.000,E1 353.742} C_DIS
LIN {X -0.012,Y -468.248,Z 618.755,A 0.000,B 0.000,C 90.000,E1 351.837} C_DIS
LIN {X 0.094,Y -470.304,Z 618.748,A 0.000,B 0.000,C 90.000,E1 350.566} C_DIS
LIN {X -0.040,Y -473.381,Z 618.737,A 0.000,B 0.000,C 90.000,E1 348.701} C_DIS
LIN {X -0.215,Y -477.717,Z 618.723,A 0.000,B 0.000,C 90.000,E1 346.228} C_DIS
LIN {X 0.032,Y -481.106,Z 618.713,A 0.000,B 0.000,C 90.000,E1 344.338} C_DIS
LIN {X 0.017,Y -485.165,Z 618.701,A 0.000,B 0.000,C 90.000,E1 342.181} C_DIS
LIN {X -0.223,Y -488.748,Z 618.691,A 0.000,B 0.000,C 90.000,E1 340.369} C_DIS
LIN {X -0.083,Y -491.693,Z 618.682,A 0.000,B 0.000,C 90.000,E1 338.827} C_DIS
LIN {X -0.068,Y -494.422,Z 618.674,A 0.000,B 0.000,C 90.000,E1 337.305} C_DIS
LIN {X -0.136,Y -496.450,Z 618.667,A 0.000,B 0.000,C 90.000,E1 336.102} C_DIS
LIN {X -0.105,Y -498.813,Z 618.659,A 0.000,B 0.000,C 90.000,E1 334.588} C_DIS
LIN {X -0.040,Y -501.090,Z 618.650,A 0.000,B 0.000,C 90.000,E1 333.076} C_DIS
LIN {X 0.077,Y -503.298,Z 618.642,A 0.000,B 0.000,C 90.000,E1 331.563} C_DIS
LIN {X -0.127,Y -505.906,Z 618.632,A 0.000,B 0.000,C 90.000,E1 329.793} C_DIS
LIN {X 0.240,Y -513.430,Z 618.609,A 0.000,B 0.000,C 90.000,E1 325.595} C_DIS
LIN {X -0.012,Y -516.974,Z 618.601,A 0.000,B 0.000,C 90.000,E1 324.149} C_DIS
LIN {X -0.080,Y -520.357,Z 618.595,A 0.000,B 0.000,C 90.000,E1 323.130} C_DIS
LIN {X 0.048,Y -521.075,Z 618.594,A 0.000,B 0.000,C 90.000,E1 322.970} C_DIS
LIN {X -0.002,Y -522.248,Z 618.593,A 0.000,B 0.000,C 90.000,E1 322.683} C_DIS
LIN {X -0.185,Y -522.960,Z 618.592,A 0.000,B 0.000,C 90.000,E1 322.557} C_DIS
LIN {X -0.232,Y -524.831,Z 618.590,A 0.000,B 0.000,C 90.000,E1 322.271} C_DIS
LIN {X -0.013,Y -527.553,Z 618.588,A 0.000,B 0.000,C 90.000,E1 321.904} C_DIS
LIN {X 0.207,Y -531.811,Z 618.586,A 0.000,B 0.000,C 90.000,E1 321.457} C_DIS
LIN {X -0.287,Y -539.253,Z 618.583,A 0.000,B 0.000,C 90.000,E1 320.884} C_DIS
LIN {X -0.092,Y -544.730,Z 618.580,A 0.000,B 0.000,C 90.000,E1 320.436} C_DIS
LIN {X -0.111,Y -557.821,Z 618.574,A 0.000,B 0.000,C 90.000,E1 319.380} C_DIS
LIN {X 0.060,Y -570.846,Z 618.569,A 0.000,B 0.000,C 90.000,E1 318.324} C_DIS
LIN {X -0.251,Y -580.854,Z 618.564,A 0.000,B 0.000,C 90.000,E1 317.553} C_DIS
LIN {X 0.053,Y -587.766,Z 618.561,A 0.000,B 0.000,C 90.000,E1 316.944} C_DIS
LIN {X -0.087,Y -593.143,Z 618.558,A 0.000,B 0.000,C 90.000,E1 316.500} C_DIS
LIN {X -0.130,Y -600.977,Z 618.555,A 0.000,B 0.000,C 90.000,E1 315.810} C_DIS
LIN {X -0.099,Y -606.113,Z 618.552,A 0.000,B 0.000,C 90.000,E1 315.324} C_DIS
LIN {X 0.032,Y -610.764,Z 618.549,A 0.000,B 0.000,C 90.000,E1 314.838} C_DIS
LIN {X -0.367,Y -616.461,Z 618.546,A 0.000,B 0.000,C 90.000,E1 314.271} C_DIS
LIN {X -0.322,Y -622.128,Z 618.542,A 0.000,B 0.000,C 90.000,E1 313.623} C_DIS
LIN {X -0.288,Y -628.442,Z 618.538,A 0.000,B 0.000,C 90.000,E1 312.852} C_DIS
LIN {X -0.055,Y -634.413,Z 618.534,A 0.000,B 0.000,C 90.000,E1 312.081} C_DIS
LIN {X -0.387,Y -641.256,Z 618.529,A 0.000,B 0.000,C 90.000,E1 311.229} C_DIS
LIN {X -0.161,Y -647.799,Z 618.524,A 0.000,B 0.000,C 90.000,E1 310.334} C_DIS
LIN {X -0.292,Y -652.109,Z 618.521,A 0.000,B 0.000,C 90.000,E1 309.725} C_DIS
LIN {X 0.094,Y -655.320,Z 618.518,A 0.000,B 0.000,C 90.000,E1 309.197} C_DIS
LIN {X 0.091,Y -658.267,Z 618.515,A 0.000,B 0.000,C 90.000,E1 308.705} C_DIS
LIN {X 0.074,Y -662.254,Z 618.511,A 0.000,B 0.000,C 90.000,E1 307.971} C_DIS
LIN {X 0.047,Y -665.373,Z 618.508,A 0.000,B 0.000,C 90.000,E1 307.363} C_DIS
LIN {X -0.315,Y -668.848,Z 618.504,A 0.000,B 0.000,C 90.000,E1 306.664} C_DIS
LIN {X 0.197,Y -669.952,Z 618.502,A 0.000,B 0.000,C 90.000,E1 306.377} C_DIS
LIN {X -0.137,Y -673.757,Z 618.497,A 0.000,B 0.000,C 90.000,E1 305.438} C_DIS
LIN {X -0.265,Y -677.348,Z 618.492,A 0.000,B 0.000,C 90.000,E1 304.485} C_DIS
LIN {X -0.167,Y -682.175,Z 618.484,A 0.000,B 0.000,C 90.000,E1 303.038} C_DIS
LIN {X 0.013,Y -686.758,Z 618.476,A 0.000,B 0.000,C 90.000,E1 301.592} C_DIS
LIN {X -0.074,Y -690.459,Z 618.469,A 0.000,B 0.000,C 90.000,E1 300.413} C_DIS
LIN {X 0.249,Y -693.953,Z 618.462,A 0.000,B 0.000,C 90.000,E1 299.205} C_DIS
LIN {X 0.024,Y -696.608,Z 618.457,A 0.000,B 0.000,C 90.000,E1 298.281} C_DIS
LIN {X 0.121,Y -699.048,Z 618.452,A 0.000,B 0.000,C 90.000,E1 297.334} C_DIS
LIN {X 0.033,Y -700.165,Z 618.449,A 0.000,B 0.000,C 90.000,E1 296.873} C_DIS
LIN {X -0.052,Y -701.023,Z 618.447,A 0.000,B 0.000,C 90.000,E1 296.411} C_DIS
LIN {X -0.168,Y -701.507,Z 618.443,A 0.000,B 0.000,C 90.000,E1 295.720} C_DIS
LIN {X 0.382,Y -700.534,Z 618.440,A 0.000,B 0.000,C 90.000,E1 295.207} C_DIS
LIN {X -0.275,Y -699.928,Z 618.439,A 0.000,B 0.000,C 90.000,E1 295.027} C_DIS
LIN {X -0.139,Y -699.326,Z 618.438,A 0.000,B 0.000,C 90.000,E1 294.899} C_DIS
LIN {X 0.392,Y -695.722,Z 618.436,A 0.000,B 0.000,C 90.000,E1 294.387} C_DIS
LIN {X -0.399,Y -694.659,Z 618.435,A 0.000,B 0.000,C 90.000,E1 294.335} C_DIS
LIN {X -0.271,Y -693.031,Z 618.434,A 0.000,B 0.000,C 90.000,E1 294.207} C_DIS
LIN {X -0.218,Y -684.161,Z 618.432,A 0.000,B 0.000,C 90.000,E1 293.823} C_DIS
LIN {X 0.043,Y -679.454,Z 618.432,A 0.000,B 0.000,C 90.000,E1 293.695} C_DIS
LIN {X 0.141,Y -673.224,Z 618.431,A 0.000,B 0.000,C 90.000,E1 293.590} C_DIS
LIN {X 0.384,Y -658.249,Z 618.430,A 0.000,B 0.000,C 90.000,E1 293.387} C_DIS
LIN {X 0.045,Y -644.741,Z 618.429,A 0.000,B 0.000,C 90.000,E1 293.206} C_DIS
LIN {X 0.008,Y -635.049,Z 618.428,A 0.000,B 0.000,C 90.000,E1 293.025} C_DIS
LIN {X 0.265,Y -625.077,Z 618.427,A 0.000,B 0.000,C 90.000,E1 292.770} C_DIS
LIN {X -0.088,Y -608.446,Z 618.424,A 0.000,B 0.000,C 90.000,E1 292.333} C_DIS
LIN {X -0.038,Y -580.846,Z 618.419,A 0.000,B 0.000,C 90.000,E1 291.461} C_DIS
LIN {X 0.163,Y -575.278,Z 618.418,A 0.000,B 0.000,C 90.000,E1 291.280} C_DIS
LIN {X 0.180,Y -566.994,Z 618.417,A 0.000,B 0.000,C 90.000,E1 291.046} C_DIS
LIN {X -0.042,Y -564.383,Z 618.417,A 0.000,B 0.000,C 90.000,E1 290.972} C_DIS
LIN {X -0.017,Y -559.576,Z 618.415,A 0.000,B 0.000,C 90.000,E1 290.737} C_DIS
LIN {X -0.160,Y -557.634,Z 618.414,A 0.000,B 0.000,C 90.000,E1 290.556} C_DIS
LIN {X -0.201,Y -557.598,Z 618.414,A 0.000,B 0.000,C 90.000,E1 290.556} C_DIS
LIN {X 0.129,Y -556.974,Z 618.413,A 0.000,B 0.000,C 90.000,E1 290.301} C_DIS
LIN {X 0.283,Y -556.793,Z 618.408,A 0.000,B 0.000,C 90.000,E1 289.450} C_DIS
LIN {X -0.087,Y -556.840,Z 618.399,A 0.000,B 0.000,C 90.000,E1 287.819} C_DIS
LIN {X 0.196,Y -556.578,Z 618.393,A 0.000,B 0.000,C 90.000,E1 286.677} C_DIS
LIN {X 0.058,Y -556.088,Z 618.385,A 0.000,B 0.000,C 90.000,E1 285.300} C_DIS
LIN {X 0.298,Y -555.450,Z 618.377,A 0.000,B 0.000,C 90.000,E1 283.883} C_DIS
LIN {X -0.010,Y -554.572,Z 618.368,A 0.000,B 0.000,C 90.000,E1 282.243} C_DIS
LIN {X 0.213,Y -553.717,Z 618.359,A 0.000,B 0.000,C 90.000,E1 280.546} C_DIS
LIN {X -0.234,Y -552.915,Z 618.349,A 0.000,B 0.000,C 90.000,E1 278.916} C_DIS
LIN {X -0.128,Y -551.989,Z 618.339,A 0.000,B 0.000,C 90.000,E1 276.947} C_DIS
LIN {X -0.221,Y -551.319,Z 618.329,A 0.000,B 0.000,C 90.000,E1 275.277} C_DIS
LIN {X 0.231,Y -550.723,Z 618.318,A 0.000,B 0.000,C 90.000,E1 273.269} C_DIS
LIN {X 0.119,Y -550.187,Z 618.307,A 0.000,B 0.000,C 90.000,E1 271.318} C_DIS
LIN {X -0.150,Y -549.780,Z 618.300,A 0.000,B 0.000,C 90.000,E1 269.943} C_DIS
LIN {X 0.121,Y -549.210,Z 618.292,A 0.000,B 0.000,C 90.000,E1 268.511} C_DIS
LIN {X -0.080,Y -548.520,Z 618.282,A 0.000,B 0.000,C 90.000,E1 266.846} C_DIS
LIN {X 0.178,Y -547.861,Z 618.275,A 0.000,B 0.000,C 90.000,E1 265.412} C_DIS
LIN {X -0.121,Y -547.191,Z 618.268,A 0.000,B 0.000,C 90.000,E1 264.318} C_DIS
LIN {X 0.114,Y -546.449,Z 618.262,A 0.000,B 0.000,C 90.000,E1 263.166} C_DIS
LIN {X -0.134,Y -545.454,Z 618.256,A 0.000,B 0.000,C 90.000,E1 262.064} C_DIS
LIN {X 0.149,Y -544.014,Z 618.248,A 0.000,B 0.000,C 90.000,E1 260.622} C_DIS
LIN {X -0.073,Y -541.297,Z 618.232,A 0.000,B 0.000,C 90.000,E1 257.813} C_DIS
LIN {X -0.146,Y -539.816,Z 618.223,A 0.000,B 0.000,C 90.000,E1 256.117} C_DIS
LIN {X -0.059,Y -538.498,Z 618.215,A 0.000,B 0.000,C 90.000,E1 254.685} C_DIS
LIN {X 0.063,Y -536.634,Z 618.205,A 0.000,B 0.000,C 90.000,E1 252.960} C_DIS
LIN {X -0.216,Y -534.917,Z 618.196,A 0.000,B 0.000,C 90.000,E1 251.275} C_DIS
LIN {X 0.219,Y -533.988,Z 618.191,A 0.000,B 0.000,C 90.000,E1 250.369} C_DIS
LIN {X -0.160,Y -532.367,Z 618.185,A 0.000,B 0.000,C 90.000,E1 249.263} C_DIS
LIN {X 0.126,Y -530.145,Z 618.177,A 0.000,B 0.000,C 90.000,E1 247.794} C_DIS
LIN {X 0.077,Y -527.599,Z 618.169,A 0.000,B 0.000,C 90.000,E1 246.357} C_DIS
LIN {X 0.122,Y -526.010,Z 618.164,A 0.000,B 0.000,C 90.000,E1 245.485} C_DIS
LIN {X -0.331,Y -524.246,Z 618.159,A 0.000,B 0.000,C 90.000,E1 244.665} C_DIS
LIN {X -0.038,Y -521.079,Z 618.151,A 0.000,B 0.000,C 90.000,E1 243.179} C_DIS
LIN {X -0.170,Y -518.507,Z 618.145,A 0.000,B 0.000,C 90.000,E1 242.025} C_DIS
LIN {X 0.014,Y -515.182,Z 618.136,A 0.000,B 0.000,C 90.000,E1 240.539} C_DIS
LIN {X -0.157,Y -511.033,Z 618.127,A 0.000,B 0.000,C 90.000,E1 238.791} C_DIS
LIN {X -0.038,Y -507.311,Z 618.118,A 0.000,B 0.000,C 90.000,E1 237.296} C_DIS
LIN {X 0.010,Y -503.416,Z 618.110,A 0.000,B 0.000,C 90.000,E1 235.801} C_DIS
LIN {X -0.150,Y -499.419,Z 618.102,A 0.000,B 0.000,C 90.000,E1 234.322} C_DIS
LIN {X -0.252,Y -492.371,Z 618.087,A 0.000,B 0.000,C 90.000,E1 231.618} C_DIS
LIN {X 0.137,Y -489.279,Z 618.080,A 0.000,B 0.000,C 90.000,E1 230.356} C_DIS
LIN {X -0.104,Y -483.877,Z 618.068,A 0.000,B 0.000,C 90.000,E1 228.243} C_DIS
LIN {X -0.091,Y -480.094,Z 618.059,A 0.000,B 0.000,C 90.000,E1 226.701} C_DIS
LIN {X 0.158,Y -474.050,Z 618.046,A 0.000,B 0.000,C 90.000,E1 224.190} C_DIS
LIN {X 0.158,Y -469.079,Z 618.034,A 0.000,B 0.000,C 90.000,E1 222.000} C_DIS
LIN {X -0.104,Y -465.629,Z 618.025,A 0.000,B 0.000,C 90.000,E1 220.458} C_DIS
LIN {X 0.274,Y -462.196,Z 618.016,A 0.000,B 0.000,C 90.000,E1 218.830} C_DIS
LIN {X 0.039,Y -458.285,Z 618.005,A 0.000,B 0.000,C 90.000,E1 216.950} C_DIS
LIN {X 0.177,Y -453.909,Z 617.993,A 0.000,B 0.000,C 90.000,E1 214.692} C_DIS
LIN {X 0.140,Y -451.002,Z 617.984,A 0.000,B 0.000,C 90.000,E1 213.086} C_DIS
LIN {X -0.060,Y -446.828,Z 617.971,A 0.000,B 0.000,C 90.000,E1 210.846} C_DIS
LIN {X -0.053,Y -442.839,Z 617.959,A 0.000,B 0.000,C 90.000,E1 208.565} C_DIS
LIN {X -0.024,Y -439.884,Z 617.950,A 0.000,B 0.000,C 90.000,E1 206.924} C_DIS
LIN {X -0.061,Y -437.018,Z 617.940,A 0.000,B 0.000,C 90.000,E1 205.283} C_DIS
LIN {X 0.250,Y -433.505,Z 617.929,A 0.000,B 0.000,C 90.000,E1 203.259} C_DIS
LIN {X 0.128,Y -430.152,Z 617.918,A 0.000,B 0.000,C 90.000,E1 201.280} C_DIS
LIN {X 0.169,Y -427.916,Z 617.911,A 0.000,B 0.000,C 90.000,E1 199.939} C_DIS
LIN {X 0.008,Y -423.633,Z 617.896,A 0.000,B 0.000,C 90.000,E1 197.275} C_DIS
LIN {X -0.136,Y -419.708,Z 617.881,A 0.000,B 0.000,C 90.000,E1 194.592} C_DIS
LIN {X -0.055,Y -417.154,Z 617.872,A 0.000,B 0.000,C 90.000,E1 192.883} C_DIS
LIN {X 0.021,Y -413.067,Z 617.856,A 0.000,B 0.000,C 90.000,E1 190.141} C_DIS
LIN {X -0.192,Y -410.759,Z 617.847,A 0.000,B 0.000,C 90.000,E1 188.454} C_DIS
LIN {X -0.107,Y -408.397,Z 617.837,A 0.000,B 0.000,C 90.000,E1 186.720} C_DIS
LIN {X -0.112,Y -405.757,Z 617.826,A 0.000,B 0.000,C 90.000,E1 184.645} C_DIS
LIN {X -0.012,Y -401.575,Z 617.805,A 0.000,B 0.000,C 90.000,E1 180.802} C_DIS
LIN {X -0.137,Y -398.366,Z 617.781,A 0.000,B 0.000,C 90.000,E1 176.617} C_DIS
LIN {X 0.161,Y -396.848,Z 617.760,A 0.000,B 0.000,C 90.000,E1 172.704} C_DIS
LIN {X -0.117,Y -396.357,Z 617.744,A 0.000,B 0.000,C 90.000,E1 169.926} C_DIS
LIN {X -0.143,Y -396.370,Z 617.726,A 0.000,B 0.000,C 90.000,E1 166.756} C_DIS
LIN {X -0.035,Y -396.831,Z 617.711,A 0.000,B 0.000,C 90.000,E1 163.921} C_DIS
LIN {X 0.124,Y -397.151,Z 617.703,A 0.000,B 0.000,C 90.000,E1 162.489} C_DIS
LIN {X -0.126,Y -397.717,Z 617.689,A 0.000,B 0.000,C 90.000,E1 160.061} C_DIS
LIN {X 0.074,Y -398.405,Z 617.677,A 0.000,B 0.000,C 90.000,E1 157.922} C_DIS
LIN {X 0.223,Y -399.099,Z 617.666,A 0.000,B 0.000,C 90.000,E1 155.793} C_DIS
LIN {X 0.025,Y -399.878,Z 617.654,A 0.000,B 0.000,C 90.000,E1 153.717} C_DIS
LIN {X -0.162,Y -400.617,Z 617.642,A 0.000,B 0.000,C 90.000,E1 151.641} C_DIS
LIN {X -0.135,Y -401.278,Z 617.631,A 0.000,B 0.000,C 90.000,E1 149.537} C_DIS
LIN {X -0.236,Y -401.895,Z 617.619,A 0.000,B 0.000,C 90.000,E1 147.454} C_DIS
LIN {X 0.117,Y -402.528,Z 617.607,A 0.000,B 0.000,C 90.000,E1 145.308} C_DIS
LIN {X 0.152,Y -403.279,Z 617.596,A 0.000,B 0.000,C 90.000,E1 143.210} C_DIS
LIN {X -0.203,Y -404.012,Z 617.584,A 0.000,B 0.000,C 90.000,E1 141.170} C_DIS
LIN {X 0.149,Y -404.628,Z 617.575,A 0.000,B 0.000,C 90.000,E1 139.380} C_DIS
LIN {X -0.095,Y -405.030,Z 617.565,A 0.000,B 0.000,C 90.000,E1 137.676} C_DIS
LIN {X 0.240,Y -405.456,Z 617.555,A 0.000,B 0.000,C 90.000,E1 135.891} C_DIS
LIN {X -0.167,Y -405.918,Z 617.544,A 0.000,B 0.000,C 90.000,E1 133.866} C_DIS
LIN {X -0.115,Y -406.416,Z 617.534,A 0.000,B 0.000,C 90.000,E1 132.123} C_DIS
LIN {X -0.147,Y -407.669,Z 617.515,A 0.000,B 0.000,C 90.000,E1 128.749} C_DIS
LIN {X 0.166,Y -409.010,Z 617.512,A 0.000,B 0.000,C 90.000,E1 128.177} C_DIS
LIN {X -0.027,Y -415.032,Z 617.501,A 0.000,B 0.000,C 90.000,E1 126.137} C_DIS
LIN {X -0.098,Y -415.970,Z 617.499,A 0.000,B 0.000,C 90.000,E1 125.804} C_DIS
LIN {X 0.010,Y -418.225,Z 617.493,A 0.000,B 0.000,C 90.000,E1 124.818} C_DIS
LIN {X -0.029,Y -418.238,Z 617.493,A 0.000,B 0.000,C 90.000,E1 124.818} C_DIS
LIN {X -0.120,Y -422.173,Z 617.492,A 0.000,B 0.000,C 90.000,E1 124.532} C_DIS
LIN {X 0.235,Y -428.479,Z 617.490,A 0.000,B 0.000,C 90.000,E1 124.119} C_DIS
LIN {X 0.083,Y -445.113,Z 617.485,A 0.000,B 0.000,C 90.000,E1 123.245} C_DIS
LIN {X 0.084,Y -455.129,Z 617.482,A 0.000,B 0.000,C 90.000,E1 122.704} C_DIS
LIN {X 0.006,Y -461.826,Z 617.480,A 0.000,B 0.000,C 90.000,E1 122.339} C_DIS
LIN {X -0.183,Y -469.889,Z 617.477,A 0.000,B 0.000,C 90.000,E1 121.878} C_DIS
LIN {X -0.110,Y -479.584,Z 617.474,A 0.000,B 0.000,C 90.000,E1 121.258} C_DIS
LIN {X -0.104,Y -485.976,Z 617.471,A 0.000,B 0.000,C 90.000,E1 120.846} C_DIS
LIN {X -0.048,Y -492.259,Z 617.469,A 0.000,B 0.000,C 90.000,E1 120.413} C_DIS
LIN {X 0.130,Y -498.465,Z 617.467,A 0.000,B 0.000,C 90.000,E1 119.951} C_DIS
LIN {X -0.076,Y -506.137,Z 617.463,A 0.000,B 0.000,C 90.000,E1 119.411} C_DIS
LIN {X 0.110,Y -516.536,Z 617.459,A 0.000,B 0.000,C 90.000,E1 118.565} C_DIS
LIN {X 0.112,Y -526.711,Z 617.454,A 0.000,B 0.000,C 90.000,E1 117.719} C_DIS
LIN {X -0.235,Y -533.666,Z 617.451,A 0.000,B 0.000,C 90.000,E1 117.129} C_DIS
LIN {X -0.234,Y -537.762,Z 617.448,A 0.000,B 0.000,C 90.000,E1 116.744} C_DIS
LIN {X -0.088,Y -542.766,Z 617.446,A 0.000,B 0.000,C 90.000,E1 116.232} C_DIS
LIN {X -0.196,Y -546.551,Z 617.444,A 0.000,B 0.000,C 90.000,E1 115.848} C_DIS
LIN {X -0.126,Y -551.847,Z 617.440,A 0.000,B 0.000,C 90.000,E1 115.207} C_DIS
LIN {X -0.089,Y -556.040,Z 617.437,A 0.000,B 0.000,C 90.000,E1 114.643} C_DIS
LIN {X -0.123,Y -560.531,Z 617.433,A 0.000,B 0.000,C 90.000,E1 113.951} C_DIS
LIN {X -0.120,Y -564.470,Z 617.429,A 0.000,B 0.000,C 90.000,E1 113.259} C_DIS
LIN {X 0.012,Y -567.227,Z 617.426,A 0.000,B 0.000,C 90.000,E1 112.695} C_DIS
LIN {X 0.130,Y -568.621,Z 617.425,A 0.000,B 0.000,C 90.000,E1 112.408} C_DIS
LIN {X 0.029,Y -573.033,Z 617.419,A 0.000,B 0.000,C 90.000,E1 111.461} C_DIS
LIN {X -0.075,Y -575.929,Z 617.416,A 0.000,B 0.000,C 90.000,E1 110.791} C_DIS
LIN {X -0.238,Y -579.139,Z 617.411,A 0.000,B 0.000,C 90.000,E1 109.993} C_DIS
LIN {X 0.177,Y -582.087,Z 617.406,A 0.000,B 0.000,C 90.000,E1 109.141} C_DIS
LIN {X 0.226,Y -583.960,Z 617.404,A 0.000,B 0.000,C 90.000,E1 108.598} C_DIS
LIN {X 0.185,Y -587.220,Z 617.398,A 0.000,B 0.000,C 90.000,E1 107.528} C_DIS
LIN {X 0.125,Y -589.448,Z 617.393,A 0.000,B 0.000,C 90.000,E1 106.732} C_DIS
LIN {X 0.166,Y -592.204,Z 617.387,A 0.000,B 0.000,C 90.000,E1 105.662} C_DIS
LIN {X -0.065,Y -600.078,Z 617.371,A 0.000,B 0.000,C 90.000,E1 102.771} C_DIS
LIN {X -0.254,Y -605.229,Z 617.361,A 0.000,B 0.000,C 90.000,E1 100.950} C_DIS
LIN {X -0.256,Y -608.144,Z 617.355,A 0.000,B 0.000,C 90.000,E1 99.905} C_DIS
LIN {X -0.214,Y -610.914,Z 617.349,A 0.000,B 0.000,C 90.000,E1 98.859} C_DIS
LIN {X -0.131,Y -614.741,Z 617.341,A 0.000,B 0.000,C 90.000,E1 97.296} C_DIS
LIN {X -0.084,Y -617.133,Z 617.335,A 0.000,B 0.000,C 90.000,E1 96.258} C_DIS
LIN {X -0.006,Y -619.324,Z 617.329,A 0.000,B 0.000,C 90.000,E1 95.220} C_DIS
LIN {X -0.211,Y -621.666,Z 617.322,A 0.000,B 0.000,C 90.000,E1 93.955} C_DIS
LIN {X 0.202,Y -623.706,Z 617.315,A 0.000,B 0.000,C 90.000,E1 92.636} C_DIS
LIN {X -0.042,Y -624.771,Z 617.311,A 0.000,B 0.000,C 90.000,E1 91.892} C_DIS
LIN {X 0.085,Y -625.988,Z 617.305,A 0.000,B 0.000,C 90.000,E1 90.859} C_DIS
LIN {X -0.133,Y -626.731,Z 617.301,A 0.000,B 0.000,C 90.000,E1 90.115} C_DIS
LIN {X 0.283,Y -627.229,Z 617.296,A 0.000,B 0.000,C 90.000,E1 89.312} C_DIS
LIN {X -0.204,Y -627.570,Z 617.291,A 0.000,B 0.000,C 90.000,E1 88.339} C_DIS
LIN {X -0.042,Y -627.699,Z 617.285,A 0.000,B 0.000,C 90.000,E1 87.306} C_DIS
LIN {X -0.159,Y -627.364,Z 617.278,A 0.000,B 0.000,C 90.000,E1 86.045} C_DIS
LIN {X 0.049,Y -626.734,Z 617.272,A 0.000,B 0.000,C 90.000,E1 85.008} C_DIS
LIN {X -0.037,Y -625.772,Z 617.265,A 0.000,B 0.000,C 90.000,E1 83.742} C_DIS
LIN {X -0.164,Y -625.057,Z 617.261,A 0.000,B 0.000,C 90.000,E1 82.989} C_DIS
LIN {X 0.243,Y -624.170,Z 617.257,A 0.000,B 0.000,C 90.000,E1 82.186} C_DIS
LIN {X 0.101,Y -623.138,Z 617.253,A 0.000,B 0.000,C 90.000,E1 81.432} C_DIS
LIN {X 0.115,Y -621.024,Z 617.245,A 0.000,B 0.000,C 90.000,E1 80.151} C_DIS
LIN {X -0.283,Y -619.134,Z 617.240,A 0.000,B 0.000,C 90.000,E1 79.162} C_DIS
LIN {X -0.337,Y -616.542,Z 617.233,A 0.000,B 0.000,C 90.000,E1 77.881} C_DIS
LIN {X -0.313,Y -613.687,Z 617.225,A 0.000,B 0.000,C 90.000,E1 76.589} C_DIS
LIN {X 0.301,Y -611.822,Z 617.221,A 0.000,B 0.000,C 90.000,E1 75.755} C_DIS
LIN {X -0.098,Y -609.306,Z 617.215,A 0.000,B 0.000,C 90.000,E1 74.755} C_DIS
LIN {X -0.054,Y -605.855,Z 617.208,A 0.000,B 0.000,C 90.000,E1 73.449} C_DIS
LIN {X -0.197,Y -602.729,Z 617.202,A 0.000,B 0.000,C 90.000,E1 72.417} C_DIS
LIN {X 0.201,Y -599.304,Z 617.196,A 0.000,B 0.000,C 90.000,E1 71.329} C_DIS
LIN {X 0.082,Y -596.328,Z 617.192,A 0.000,B 0.000,C 90.000,E1 70.550} C_DIS
LIN {X -0.181,Y -591.930,Z 617.186,A 0.000,B 0.000,C 90.000,E1 69.518} C_DIS
LIN {X 0.150,Y -589.678,Z 617.183,A 0.000,B 0.000,C 90.000,E1 68.954} C_DIS
LIN {X 0.072,Y -585.413,Z 617.178,A 0.000,B 0.000,C 90.000,E1 68.028} C_DIS
LIN {X 0.017,Y -581.421,Z 617.174,A 0.000,B 0.000,C 90.000,E1 67.230} C_DIS
LIN {X -0.103,Y -576.458,Z 617.168,A 0.000,B 0.000,C 90.000,E1 66.305} C_DIS
LIN {X 0.194,Y -574.123,Z 617.166,A 0.000,B 0.000,C 90.000,E1 65.869} C_DIS
LIN {X -0.206,Y -569.927,Z 617.162,A 0.000,B 0.000,C 90.000,E1 65.229} C_DIS
LIN {X 0.221,Y -565.421,Z 617.159,A 0.000,B 0.000,C 90.000,E1 64.537} C_DIS
LIN {X 0.056,Y -560.527,Z 617.155,A 0.000,B 0.000,C 90.000,E1 63.896} C_DIS
LIN {X 0.154,Y -556.136,Z 617.152,A 0.000,B 0.000,C 90.000,E1 63.332} C_DIS
LIN {X 0.085,Y -552.436,Z 617.150,A 0.000,B 0.000,C 90.000,E1 62.922} C_DIS
LIN {X -0.212,Y -547.120,Z 617.147,A 0.000,B 0.000,C 90.000,E1 62.410} C_DIS
LIN {X -0.207,Y -541.428,Z 617.144,A 0.000,B 0.000,C 90.000,E1 61.897} C_DIS
LIN {X 0.202,Y -535.247,Z 617.141,A 0.000,B 0.000,C 90.000,E1 61.385} C_DIS
LIN {X 0.264,Y -530.504,Z 617.139,A 0.000,B 0.000,C 90.000,E1 61.051} C_DIS
LIN {X 0.064,Y -523.653,Z 617.137,A 0.000,B 0.000,C 90.000,E1 60.667} C_DIS
LIN {X 0.095,Y -518.662,Z 617.136,A 0.000,B 0.000,C 90.000,E1 60.383} C_DIS
LIN {X -0.004,Y -508.432,Z 617.133,A 0.000,B 0.000,C 90.000,E1 59.871} C_DIS
LIN {X 0.160,Y -496.432,Z 617.130,A 0.000,B 0.000,C 90.000,E1 59.282} C_DIS
LIN {X -0.009,Y -479.630,Z 617.125,A 0.000,B 0.000,C 90.000,E1 58.486} C_DIS
LIN {X 0.248,Y -459.508,Z 617.119,A 0.000,B 0.000,C 90.000,E1 57.454} C_DIS
LIN {X -0.060,Y -449.489,Z 617.116,A 0.000,B 0.000,C 90.000,E1 56.962} C_DIS
LIN {X -0.089,Y -444.325,Z 617.115,A 0.000,B 0.000,C 90.000,E1 56.707} C_DIS
LIN {X -0.131,Y -444.292,Z 617.115,A 0.000,B 0.000,C 90.000,E1 56.707} C_DIS
LIN {X -0.122,Y -443.406,Z 617.113,A 0.000,B 0.000,C 90.000,E1 56.294} C_DIS
LIN {X -0.133,Y -434.353,Z 617.091,A 0.000,B 0.000,C 90.000,E1 52.351} C_DIS
LIN {X -0.017,Y -431.854,Z 617.083,A 0.000,B 0.000,C 90.000,E1 51.009} C_DIS
LIN {X -0.031,Y -431.165,Z 617.082,A 0.000,B 0.000,C 90.000,E1 50.678} C_DIS
LIN {X 0.193,Y -428.239,Z 617.075,A 0.000,B 0.000,C 90.000,E1 49.461} C_DIS
LIN {X 0.014,Y -429.116,Z 617.067,A 0.000,B 0.000,C 90.000,E1 48.000} C_DIS
LIN {X 0.184,Y -430.002,Z 617.056,A 0.000,B 0.000,C 90.000,E1 45.972} C_DIS
LIN {X -0.247,Y -430.841,Z 617.044,A 0.000,B 0.000,C 90.000,E1 44.028} C_DIS
LIN {X 0.033,Y -431.671,Z 617.035,A 0.000,B 0.000,C 90.000,E1 42.324} C_DIS
LIN {X -0.020,Y -432.630,Z 617.024,A 0.000,B 0.000,C 90.000,E1 40.334} C_DIS
LIN {X -0.001,Y -433.569,Z 617.013,A 0.000,B 0.000,C 90.000,E1 38.338} C_DIS
LIN {X 0.106,Y -434.140,Z 617.006,A 0.000,B 0.000,C 90.000,E1 36.996} C_DIS
LIN {X -0.045,Y -434.765,Z 616.996,A 0.000,B 0.000,C 90.000,E1 35.358} C_DIS
LIN {X -0.078,Y -435.301,Z 616.987,A 0.000,B 0.000,C 90.000,E1 33.706} C_DIS
LIN {X -0.102,Y -435.699,Z 616.978,A 0.000,B 0.000,C 90.000,E1 32.054} C_DIS
LIN {X 0.044,Y -436.255,Z 616.967,A 0.000,B 0.000,C 90.000,E1 30.050} C_DIS
LIN {X -0.201,Y -436.939,Z 616.954,A 0.000,B 0.000,C 90.000,E1 27.769} C_DIS
LIN {X -0.089,Y -437.437,Z 616.945,A 0.000,B 0.000,C 90.000,E1 26.104} C_DIS
LIN {X 0.097,Y -438.210,Z 616.932,A 0.000,B 0.000,C 90.000,E1 23.770} C_DIS
LIN {X 0.124,Y -439.102,Z 616.919,A 0.000,B 0.000,C 90.000,E1 21.461} C_DIS
LIN {X 0.157,Y -439.839,Z 616.910,A 0.000,B 0.000,C 90.000,E1 19.812} C_DIS
LIN {X 0.162,Y -440.831,Z 616.897,A 0.000,B 0.000,C 90.000,E1 17.511} C_DIS
LIN {X 0.078,Y -442.220,Z 616.883,A 0.000,B 0.000,C 90.000,E1 14.898} C_DIS
LIN {X 0.098,Y -444.004,Z 616.867,A 0.000,B 0.000,C 90.000,E1 11.951} C_DIS
LIN {X 0.072,Y -445.685,Z 616.854,A 0.000,B 0.000,C 90.000,E1 9.670} C_DIS
LIN {X 0.013,Y -447.065,Z 616.845,A 0.000,B 0.000,C 90.000,E1 8.049} C_DIS
LIN {X -0.147,Y -449.143,Z 616.832,A 0.000,B 0.000,C 90.000,E1 5.796} C_DIS
LIN {X -0.185,Y -451.759,Z 616.818,A 0.000,B 0.000,C 90.000,E1 3.212} C_DIS
LIN {X -0.160,Y -454.792,Z 616.803,A 0.000,B 0.000,C 90.000,E1 0.630} C_DIS
LIN {X 0.183,Y -458.036,Z 616.790,A 0.000,B 0.000,C 90.000,E1 358.167} C_DIS
LIN {X 0.201,Y -461.468,Z 616.778,A 0.000,B 0.000,C 90.000,E1 355.931} C_DIS
LIN {X 0.182,Y -465.679,Z 616.763,A 0.000,B 0.000,C 90.000,E1 353.394} C_DIS
LIN {X 0.000,Y -468.346,Z 616.755,A 0.000,B 0.000,C 90.000,E1 351.837} C_DIS
LIN {X -0.074,Y -470.856,Z 616.746,A 0.000,B 0.000,C 90.000,E1 350.274} C_DIS
LIN {X -0.025,Y -473.446,Z 616.737,A 0.000,B 0.000,C 90.000,E1 348.701} C_DIS
LIN {X 0.109,Y -478.344,Z 616.722,A 0.000,B 0.000,C 90.000,E1 345.880} C_DIS
LIN {X -0.116,Y -482.313,Z 616.710,A 0.000,B 0.000,C 90.000,E1 343.740} C_DIS
LIN {X -0.102,Y -486.395,Z 616.698,A 0.000,B 0.000,C 90.000,E1 341.583} C_DIS
LIN {X -0.155,Y -489.970,Z 616.687,A 0.000,B 0.000,C 90.000,E1 339.752} C_DIS
LIN {X -0.204,Y -492.294,Z 616.681,A 0.000,B 0.000,C 90.000,E1 338.539} C_DIS
LIN {X 0.193,Y -494.984,Z 616.672,A 0.000,B 0.000,C 90.000,E1 336.975} C_DIS
LIN {X -0.113,Y -496.498,Z 616.667,A 0.000,B 0.000,C 90.000,E1 336.102} C_DIS
LIN {X -0.081,Y -498.844,Z 616.659,A 0.000,B 0.000,C 90.000,E1 334.588} C_DIS
LIN {X -0.014,Y -501.117,Z 616.650,A 0.000,B 0.000,C 90.000,E1 333.076} C_DIS
LIN {X 0.103,Y -503.325,Z 616.642,A 0.000,B 0.000,C 90.000,E1 331.563} C_DIS
LIN {X -0.101,Y -505.932,Z 616.632,A 0.000,B 0.000,C 90.000,E1 329.793} C_DIS
LIN {X 0.052,Y -507.759,Z 616.626,A 0.000,B 0.000,C 90.000,E1 328.584} C_DIS
LIN {X 0.185,Y -513.957,Z 616.607,A 0.000,B 0.000,C 90.000,E1 325.308} C_DIS
LIN {X -0.058,Y -517.424,Z 616.599,A 0.000,B 0.000,C 90.000,E1 323.863} C_DIS
LIN {X -0.122,Y -519.315,Z 616.596,A 0.000,B 0.000,C 90.000,E1 323.290} C_DIS
LIN {X 0.131,Y -520.109,Z 616.594,A 0.000,B 0.000,C 90.000,E1 322.970} C_DIS
LIN {X 0.152,Y -520.957,Z 616.593,A 0.000,B 0.000,C 90.000,E1 322.763} C_DIS
LIN {X -0.085,Y -522.477,Z 616.591,A 0.000,B 0.000,C 90.000,E1 322.351} C_DIS
LIN {X 0.186,Y -524.316,Z 616.589,A 0.000,B 0.000,C 90.000,E1 321.984} C_DIS
LIN {X 0.291,Y -527.749,Z 616.587,A 0.000,B 0.000,C 90.000,E1 321.537} C_DIS
LIN {X -0.153,Y -532.015,Z 616.584,A 0.000,B 0.000,C 90.000,E1 321.170} C_DIS
LIN {X -0.205,Y -537.360,Z 616.582,A 0.000,B 0.000,C 90.000,E1 320.723} C_DIS
LIN {X -0.015,Y -552.819,Z 616.575,A 0.000,B 0.000,C 90.000,E1 319.461} C_DIS
LIN {X 0.124,Y -565.849,Z 616.569,A 0.000,B 0.000,C 90.000,E1 318.405} C_DIS
LIN {X 0.154,Y -581.698,Z 616.562,A 0.000,B 0.000,C 90.000,E1 317.148} C_DIS
LIN {X 0.030,Y -587.274,Z 616.560,A 0.000,B 0.000,C 90.000,E1 316.701} C_DIS
LIN {X 0.240,Y -595.579,Z 616.556,A 0.000,B 0.000,C 90.000,E1 315.972} C_DIS
LIN {X 0.116,Y -602.018,Z 616.552,A 0.000,B 0.000,C 90.000,E1 315.405} C_DIS
LIN {X -0.293,Y -605.862,Z 616.550,A 0.000,B 0.000,C 90.000,E1 315.081} C_DIS
LIN {X -0.337,Y -608.424,Z 616.549,A 0.000,B 0.000,C 90.000,E1 314.838} C_DIS
LIN {X -0.186,Y -614.538,Z 616.545,A 0.000,B 0.000,C 90.000,E1 314.190} C_DIS
LIN {X -0.067,Y -619.201,Z 616.543,A 0.000,B 0.000,C 90.000,E1 313.662} C_DIS
LIN {X 0.000,Y -624.758,Z 616.539,A 0.000,B 0.000,C 90.000,E1 313.014} C_DIS
LIN {X 0.078,Y -632.969,Z 616.533,A 0.000,B 0.000,C 90.000,E1 312.000} C_DIS
LIN {X 0.131,Y -640.834,Z 616.528,A 0.000,B 0.000,C 90.000,E1 310.987} C_DIS
LIN {X -0.061,Y -646.513,Z 616.524,A 0.000,B 0.000,C 90.000,E1 310.253} C_DIS
LIN {X -0.205,Y -650.951,Z 616.520,A 0.000,B 0.000,C 90.000,E1 309.644} C_DIS
LIN {X 0.193,Y -654.978,Z 616.517,A 0.000,B 0.000,C 90.000,E1 308.991} C_DIS
LIN {X 0.113,Y -658.613,Z 616.513,A 0.000,B 0.000,C 90.000,E1 308.382} C_DIS
LIN {X -0.349,Y -661.973,Z 616.510,A 0.000,B 0.000,C 90.000,E1 307.810} C_DIS
LIN {X 0.145,Y -665.100,Z 616.507,A 0.000,B 0.000,C 90.000,E1 307.156} C_DIS
LIN {X -0.214,Y -668.553,Z 616.503,A 0.000,B 0.000,C 90.000,E1 306.457} C_DIS
LIN {X -0.149,Y -671.623,Z 616.498,A 0.000,B 0.000,C 90.000,E1 305.724} C_DIS
LIN {X 0.081,Y -675.285,Z 616.493,A 0.000,B 0.000,C 90.000,E1 304.739} C_DIS
LIN {X -0.023,Y -678.699,Z 616.488,A 0.000,B 0.000,C 90.000,E1 303.785} C_DIS
LIN {X -0.259,Y -681.151,Z 616.484,A 0.000,B 0.000,C 90.000,E1 303.086} C_DIS
LIN {X 0.116,Y -685.807,Z 616.476,A 0.000,B 0.000,C 90.000,E1 301.623} C_DIS
LIN {X -0.220,Y -689.554,Z 616.469,A 0.000,B 0.000,C 90.000,E1 300.463} C_DIS
LIN {X -0.257,Y -693.138,Z 616.463,A 0.000,B 0.000,C 90.000,E1 299.283} C_DIS
LIN {X 0.122,Y -695.858,Z 616.457,A 0.000,B 0.000,C 90.000,E1 298.309} C_DIS
LIN {X -0.079,Y -698.381,Z 616.452,A 0.000,B 0.000,C 90.000,E1 297.385} C_DIS
LIN {X 0.094,Y -700.037,Z 616.448,A 0.000,B 0.000,C 90.000,E1 296.668} C_DIS
LIN {X 0.051,Y -700.471,Z 616.447,A 0.000,B 0.000,C 90.000,E1 296.437} C_DIS
LIN {X 0.242,Y -701.007,Z 616.443,A 0.000,B 0.000,C 90.000,E1 295.720} C_DIS
LIN {X -0.143,Y -700.088,Z 616.440,A 0.000,B 0.000,C 90.000,E1 295.283} C_DIS
LIN {X 0.129,Y -699.504,Z 616.439,A 0.000,B 0.000,C 90.000,E1 295.027} C_DIS
LIN {X 0.264,Y -698.937,Z 616.438,A 0.000,B 0.000,C 90.000,E1 294.899} C_DIS
LIN {X 0.186,Y -694.570,Z 616.435,A 0.000,B 0.000,C 90.000,E1 294.335} C_DIS
LIN {X 0.313,Y -693.135,Z 616.435,A 0.000,B 0.000,C 90.000,E1 294.207} C_DIS
LIN {X -0.192,Y -690.749,Z 616.434,A 0.000,B 0.000,C 90.000,E1 294.131} C_DIS
LIN {X -0.133,Y -685.529,Z 616.433,A 0.000,B 0.000,C 90.000,E1 293.898} C_DIS
LIN {X -0.087,Y -683.685,Z 616.432,A 0.000,B 0.000,C 90.000,E1 293.823} C_DIS
LIN {X -0.112,Y -677.662,Z 616.432,A 0.000,B 0.000,C 90.000,E1 293.695} C_DIS
LIN {X -0.350,Y -673.005,Z 616.431,A 0.000,B 0.000,C 90.000,E1 293.643} C_DIS
LIN {X -0.112,Y -658.157,Z 616.430,A 0.000,B 0.000,C 90.000,E1 293.439} C_DIS
LIN {X 0.118,Y -644.450,Z 616.429,A 0.000,B 0.000,C 90.000,E1 293.206} C_DIS
LIN {X 0.091,Y -634.859,Z 616.428,A 0.000,B 0.000,C 90.000,E1 293.025} C_DIS
LIN {X -0.234,Y -624.896,Z 616.427,A 0.000,B 0.000,C 90.000,E1 292.823} C_DIS
LIN {X -0.050,Y -608.185,Z 616.424,A 0.000,B 0.000,C 90.000,E1 292.333} C_DIS
LIN {X -0.189,Y -584.099,Z 616.420,A 0.000,B 0.000,C 90.000,E1 291.589} C_DIS
LIN {X -0.054,Y -576.862,Z 616.419,A 0.000,B 0.000,C 90.000,E1 291.354} C_DIS
LIN {X 0.257,Y -564.813,Z 616.417,A 0.000,B 0.000,C 90.000,E1 290.972} C_DIS
LIN {X 0.076,Y -559.645,Z 616.415,A 0.000,B 0.000,C 90.000,E1 290.737} C_DIS
LIN {X 0.053,Y -557.824,Z 616.414,A 0.000,B 0.000,C 90.000,E1 290.556} C_DIS
LIN {X 0.013,Y -557.785,Z 616.414,A 0.000,B 0.000,C 90.000,E1 290.556} C_DIS
LIN {X 0.052,Y -557.227,Z 616.413,A 0.000,B 0.000,C 90.000,E1 290.355} C_DIS
LIN {X 0.157,Y -557.021,Z 616.412,A 0.000,B 0.000,C 90.000,E1 290.066} C_DIS
LIN {X 0.090,Y -556.981,Z 616.401,A 0.000,B 0.000,C 90.000,E1 288.127} C_DIS
LIN {X -0.152,Y -556.841,Z 616.395,A 0.000,B 0.000,C 90.000,E1 287.040} C_DIS
LIN {X 0.254,Y -556.345,Z 616.387,A 0.000,B 0.000,C 90.000,E1 285.607} C_DIS
LIN {X -0.032,Y -555.743,Z 616.379,A 0.000,B 0.000,C 90.000,E1 284.245} C_DIS
LIN {X -0.074,Y -554.726,Z 616.368,A 0.000,B 0.000,C 90.000,E1 282.299} C_DIS
LIN {X 0.149,Y -553.871,Z 616.359,A 0.000,B 0.000,C 90.000,E1 280.602} C_DIS
LIN {X 0.249,Y -553.036,Z 616.350,A 0.000,B 0.000,C 90.000,E1 278.916} C_DIS
LIN {X -0.190,Y -552.109,Z 616.339,A 0.000,B 0.000,C 90.000,E1 277.004} C_DIS
LIN {X 0.164,Y -551.567,Z 616.331,A 0.000,B 0.000,C 90.000,E1 275.568} C_DIS
LIN {X 0.257,Y -550.761,Z 616.317,A 0.000,B 0.000,C 90.000,E1 273.037} C_DIS
LIN {X 0.173,Y -550.158,Z 616.305,A 0.000,B 0.000,C 90.000,E1 270.802} C_DIS
LIN {X -0.096,Y -549.676,Z 616.297,A 0.000,B 0.000,C 90.000,E1 269.427} C_DIS
LIN {X 0.188,Y -549.072,Z 616.289,A 0.000,B 0.000,C 90.000,E1 267.993} C_DIS
LIN {X -0.084,Y -548.528,Z 616.281,A 0.000,B 0.000,C 90.000,E1 266.617} C_DIS
LIN {X 0.217,Y -547.862,Z 616.273,A 0.000,B 0.000,C 90.000,E1 265.179} C_DIS
LIN {X -0.133,Y -547.161,Z 616.267,A 0.000,B 0.000,C 90.000,E1 264.090} C_DIS
LIN {X 0.074,Y -546.614,Z 616.262,A 0.000,B 0.000,C 90.000,E1 263.223} C_DIS
LIN {X 0.277,Y -545.898,Z 616.258,A 0.000,B 0.000,C 90.000,E1 262.356} C_DIS
LIN {X 0.029,Y -544.507,Z 616.250,A 0.000,B 0.000,C 90.000,E1 260.971} C_DIS
LIN {X -0.068,Y -543.041,Z 616.242,A 0.000,B 0.000,C 90.000,E1 259.567} C_DIS
LIN {X -0.128,Y -541.251,Z 616.231,A 0.000,B 0.000,C 90.000,E1 257.589} C_DIS
LIN {X -0.157,Y -539.989,Z 616.223,A 0.000,B 0.000,C 90.000,E1 256.172} C_DIS
LIN {X -0.206,Y -538.670,Z 616.215,A 0.000,B 0.000,C 90.000,E1 254.755} C_DIS
LIN {X 0.066,Y -536.810,Z 616.206,A 0.000,B 0.000,C 90.000,E1 253.015} C_DIS
LIN {X -0.204,Y -535.092,Z 616.196,A 0.000,B 0.000,C 90.000,E1 251.329} C_DIS
LIN {X 0.237,Y -534.163,Z 616.191,A 0.000,B 0.000,C 90.000,E1 250.423} C_DIS
LIN {X 0.160,Y -533.013,Z 616.187,A 0.000,B 0.000,C 90.000,E1 249.571} C_DIS
LIN {X -0.036,Y -530.799,Z 616.179,A 0.000,B 0.000,C 90.000,E1 248.156} C_DIS
LIN {X 0.028,Y -528.784,Z 616.172,A 0.000,B 0.000,C 90.000,E1 246.997} C_DIS
LIN {X 0.166,Y -526.173,Z 616.164,A 0.000,B 0.000,C 90.000,E1 245.537} C_DIS
LIN {X -0.121,Y -523.768,Z 616.158,A 0.000,B 0.000,C 90.000,E1 244.409} C_DIS
LIN {X -0.216,Y -521.247,Z 616.151,A 0.000,B 0.000,C 90.000,E1 243.256} C_DIS
LIN {X -0.105,Y -518.672,Z 616.145,A 0.000,B 0.000,C 90.000,E1 242.076} C_DIS
LIN {X 0.087,Y -515.342,Z 616.137,A 0.000,B 0.000,C 90.000,E1 240.589} C_DIS
LIN {X 0.098,Y -511.191,Z 616.127,A 0.000,B 0.000,C 90.000,E1 238.820} C_DIS
LIN {X -0.121,Y -508.207,Z 616.120,A 0.000,B 0.000,C 90.000,E1 237.661} C_DIS
LIN {X -0.063,Y -504.353,Z 616.112,A 0.000,B 0.000,C 90.000,E1 236.167} C_DIS
LIN {X -0.095,Y -501.136,Z 616.105,A 0.000,B 0.000,C 90.000,E1 234.975} C_DIS
LIN {X 0.130,Y -495.491,Z 616.094,A 0.000,B 0.000,C 90.000,E1 232.844} C_DIS
LIN {X -0.040,Y -490.955,Z 616.084,A 0.000,B 0.000,C 90.000,E1 231.045} C_DIS
LIN {X -0.243,Y -485.472,Z 616.072,A 0.000,B 0.000,C 90.000,E1 228.933} C_DIS
LIN {X -0.064,Y -480.922,Z 616.061,A 0.000,B 0.000,C 90.000,E1 227.067} C_DIS
LIN {X -0.118,Y -474.852,Z 616.048,A 0.000,B 0.000,C 90.000,E1 224.595} C_DIS
LIN {X -0.008,Y -469.131,Z 616.034,A 0.000,B 0.000,C 90.000,E1 222.081} C_DIS
LIN {X -0.267,Y -465.655,Z 616.025,A 0.000,B 0.000,C 90.000,E1 220.539} C_DIS
LIN {X 0.114,Y -462.226,Z 616.016,A 0.000,B 0.000,C 90.000,E1 218.910} C_DIS
LIN {X -0.116,Y -458.320,Z 616.006,A 0.000,B 0.000,C 90.000,E1 217.030} C_DIS
LIN {X 0.101,Y -452.754,Z 615.990,A 0.000,B 0.000,C 90.000,E1 214.119} C_DIS
LIN {X -0.210,Y -449.797,Z 615.981,A 0.000,B 0.000,C 90.000,E1 212.546} C_DIS
LIN {X -0.126,Y -446.238,Z 615.970,A 0.000,B 0.000,C 90.000,E1 210.590} C_DIS
LIN {X 0.081,Y -442.279,Z 615.957,A 0.000,B 0.000,C 90.000,E1 208.281} C_DIS
LIN {X 0.151,Y -438.182,Z 615.944,A 0.000,B 0.000,C 90.000,E1 205.976} C_DIS
LIN {X -0.081,Y -434.126,Z 615.932,A 0.000,B 0.000,C 90.000,E1 203.695} C_DIS
LIN {X 0.030,Y -430.186,Z 615.919,A 0.000,B 0.000,C 90.000,E1 201.354} C_DIS
LIN {X 0.027,Y -427.399,Z 615.909,A 0.000,B 0.000,C 90.000,E1 199.685} C_DIS
LIN {X 0.057,Y -423.690,Z 615.896,A 0.000,B 0.000,C 90.000,E1 197.330} C_DIS
LIN {X -0.091,Y -419.789,Z 615.881,A 0.000,B 0.000,C 90.000,E1 194.647} C_DIS
LIN {X -0.012,Y -417.238,Z 615.872,A 0.000,B 0.000,C 90.000,E1 192.939} C_DIS
LIN {X 0.063,Y -413.154,Z 615.857,A 0.000,B 0.000,C 90.000,E1 190.197} C_DIS
LIN {X -0.151,Y -410.846,Z 615.847,A 0.000,B 0.000,C 90.000,E1 188.511} C_DIS
LIN {X -0.067,Y -408.515,Z 615.838,A 0.000,B 0.000,C 90.000,E1 186.777} C_DIS
LIN {X -0.100,Y -405.427,Z 615.824,A 0.000,B 0.000,C 90.000,E1 184.359} C_DIS
LIN {X -0.005,Y -401.375,Z 615.803,A 0.000,B 0.000,C 90.000,E1 180.516} C_DIS
LIN {X -0.141,Y -398.282,Z 615.780,A 0.000,B 0.000,C 90.000,E1 176.331} C_DIS
LIN {X -0.174,Y -396.950,Z 615.760,A 0.000,B 0.000,C 90.000,E1 172.818} C_DIS
LIN {X -0.053,Y -396.457,Z 615.744,A 0.000,B 0.000,C 90.000,E1 169.982} C_DIS
LIN {X -0.162,Y -396.460,Z 615.727,A 0.000,B 0.000,C 90.000,E1 166.825} C_DIS
LIN {X 0.045,Y -396.950,Z 615.711,A 0.000,B 0.000,C 90.000,E1 163.976} C_DIS
LIN {X -0.169,Y -397.263,Z 615.703,A 0.000,B 0.000,C 90.000,E1 162.598} C_DIS
LIN {X -0.033,Y -397.844,Z 615.690,A 0.000,B 0.000,C 90.000,E1 160.115} C_DIS
LIN {X 0.177,Y -398.544,Z 615.678,A 0.000,B 0.000,C 90.000,E1 157.975} C_DIS
LIN {X -0.191,Y -399.250,Z 615.666,A 0.000,B 0.000,C 90.000,E1 155.921} C_DIS
LIN {X 0.148,Y -400.058,Z 615.654,A 0.000,B 0.000,C 90.000,E1 153.768} C_DIS
LIN {X -0.027,Y -400.816,Z 615.643,A 0.000,B 0.000,C 90.000,E1 151.691} C_DIS
LIN {X 0.011,Y -401.483,Z 615.631,A 0.000,B 0.000,C 90.000,E1 149.587} C_DIS
LIN {X -0.076,Y -402.099,Z 615.619,A 0.000,B 0.000,C 90.000,E1 147.502} C_DIS
LIN {X -0.057,Y -402.630,Z 615.610,A 0.000,B 0.000,C 90.000,E1 145.754} C_DIS
LIN {X 0.212,Y -403.323,Z 615.598,A 0.000,B 0.000,C 90.000,E1 143.623} C_DIS
LIN {X 0.180,Y -404.042,Z 615.586,A 0.000,B 0.000,C 90.000,E1 141.537} C_DIS
LIN {X -0.036,Y -404.650,Z 615.577,A 0.000,B 0.000,C 90.000,E1 139.828} C_DIS
LIN {X 0.059,Y -404.951,Z 615.571,A 0.000,B 0.000,C 90.000,E1 138.771} C_DIS
LIN {X -0.049,Y -405.424,Z 615.559,A 0.000,B 0.000,C 90.000,E1 136.701} C_DIS
LIN {X -0.134,Y -405.730,Z 615.552,A 0.000,B 0.000,C 90.000,E1 135.324} C_DIS
LIN {X 0.171,Y -406.319,Z 615.538,A 0.000,B 0.000,C 90.000,E1 132.852} C_DIS
LIN {X 0.100,Y -406.839,Z 615.527,A 0.000,B 0.000,C 90.000,E1 130.782} C_DIS
LIN {X 0.091,Y -407.669,Z 615.515,A 0.000,B 0.000,C 90.000,E1 128.705} C_DIS
LIN {X -0.026,Y -415.562,Z 615.500,A 0.000,B 0.000,C 90.000,E1 125.964} C_DIS
LIN {X -0.047,Y -418.936,Z 615.492,A 0.000,B 0.000,C 90.000,E1 124.532} C_DIS
LIN {X -0.086,Y -418.977,Z 615.492,A 0.000,B 0.000,C 90.000,E1 124.532} C_DIS
LIN {X 0.063,Y -422.676,Z 615.490,A 0.000,B 0.000,C 90.000,E1 124.246} C_DIS
LIN {X -0.142,Y -427.493,Z 615.489,A 0.000,B 0.000,C 90.000,E1 123.992} C_DIS
LIN {X -0.086,Y -432.861,Z 615.487,A 0.000,B 0.000,C 90.000,E1 123.706} C_DIS
LIN {X -0.088,Y -449.934,Z 615.482,A 0.000,B 0.000,C 90.000,E1 122.801} C_DIS
LIN {X 0.148,Y -461.556,Z 615.479,A 0.000,B 0.000,C 90.000,E1 122.133} C_DIS
LIN {X -0.116,Y -466.494,Z 615.477,A 0.000,B 0.000,C 90.000,E1 121.878} C_DIS
LIN {X -0.092,Y -477.801,Z 615.473,A 0.000,B 0.000,C 90.000,E1 121.180} C_DIS
LIN {X 0.002,Y -485.651,Z 615.470,A 0.000,B 0.000,C 90.000,E1 120.669} C_DIS
LIN {X 0.170,Y -490.379,Z 615.469,A 0.000,B 0.000,C 90.000,E1 120.335} C_DIS
LIN {X -0.002,Y -496.567,Z 615.466,A 0.000,B 0.000,C 90.000,E1 119.922} C_DIS
LIN {X 0.240,Y -504.423,Z 615.463,A 0.000,B 0.000,C 90.000,E1 119.333} C_DIS
LIN {X 0.028,Y -512.942,Z 615.459,A 0.000,B 0.000,C 90.000,E1 118.693} C_DIS
LIN {X -0.087,Y -518.851,Z 615.457,A 0.000,B 0.000,C 90.000,E1 118.231} C_DIS
LIN {X 0.090,Y -525.835,Z 615.454,A 0.000,B 0.000,C 90.000,E1 117.641} C_DIS
LIN {X 0.253,Y -531.485,Z 615.451,A 0.000,B 0.000,C 90.000,E1 117.129} C_DIS
LIN {X 0.291,Y -535.744,Z 615.449,A 0.000,B 0.000,C 90.000,E1 116.744} C_DIS
LIN {X 0.297,Y -541.087,Z 615.446,A 0.000,B 0.000,C 90.000,E1 116.232} C_DIS
LIN {X 0.290,Y -546.060,Z 615.443,A 0.000,B 0.000,C 90.000,E1 115.720} C_DIS
LIN {X 0.122,Y -548.398,Z 615.442,A 0.000,B 0.000,C 90.000,E1 115.463} C_DIS
LIN {X -0.287,Y -550.487,Z 615.440,A 0.000,B 0.000,C 90.000,E1 115.283} C_DIS
LIN {X 0.033,Y -552.522,Z 615.439,A 0.000,B 0.000,C 90.000,E1 114.975} C_DIS
LIN {X 0.217,Y -555.502,Z 615.437,A 0.000,B 0.000,C 90.000,E1 114.591} C_DIS
LIN {X 0.182,Y -560.166,Z 615.433,A 0.000,B 0.000,C 90.000,E1 113.898} C_DIS
LIN {X 0.188,Y -564.201,Z 615.429,A 0.000,B 0.000,C 90.000,E1 113.206} C_DIS
LIN {X 0.132,Y -568.510,Z 615.424,A 0.000,B 0.000,C 90.000,E1 112.386} C_DIS
LIN {X -0.100,Y -572.381,Z 615.420,A 0.000,B 0.000,C 90.000,E1 111.589} C_DIS
LIN {X -0.208,Y -575.408,Z 615.416,A 0.000,B 0.000,C 90.000,E1 110.918} C_DIS
LIN {X 0.171,Y -578.703,Z 615.412,A 0.000,B 0.000,C 90.000,E1 110.066} C_DIS
LIN {X -0.121,Y -582.665,Z 615.406,A 0.000,B 0.000,C 90.000,E1 109.014} C_DIS
LIN {X -0.071,Y -584.549,Z 615.403,A 0.000,B 0.000,C 90.000,E1 108.471} C_DIS
LIN {X 0.221,Y -587.053,Z 615.398,A 0.000,B 0.000,C 90.000,E1 107.638} C_DIS
LIN {X -0.334,Y -590.085,Z 615.392,A 0.000,B 0.000,C 90.000,E1 106.622} C_DIS
LIN {X -0.123,Y -592.832,Z 615.386,A 0.000,B 0.000,C 90.000,E1 105.536} C_DIS
LIN {X 0.242,Y -600.862,Z 615.370,A 0.000,B 0.000,C 90.000,E1 102.591} C_DIS
LIN {X -0.047,Y -606.100,Z 615.360,A 0.000,B 0.000,C 90.000,E1 100.782} C_DIS
LIN {X -0.292,Y -609.723,Z 615.353,A 0.000,B 0.000,C 90.000,E1 99.500} C_DIS
LIN {X 0.124,Y -611.776,Z 615.348,A 0.000,B 0.000,C 90.000,E1 98.681} C_DIS
LIN {X -0.134,Y -615.064,Z 615.341,A 0.000,B 0.000,C 90.000,E1 97.409} C_DIS
LIN {X -0.087,Y -617.498,Z 615.335,A 0.000,B 0.000,C 90.000,E1 96.372} C_DIS
LIN {X -0.006,Y -619.761,Z 615.330,A 0.000,B 0.000,C 90.000,E1 95.334} C_DIS
LIN {X 0.116,Y -622.606,Z 615.321,A 0.000,B 0.000,C 90.000,E1 93.784} C_DIS
LIN {X -0.075,Y -624.639,Z 615.314,A 0.000,B 0.000,C 90.000,E1 92.522} C_DIS
LIN {X -0.234,Y -626.335,Z 615.307,A 0.000,B 0.000,C 90.000,E1 91.260} C_DIS
LIN {X -0.102,Y -627.372,Z 615.301,A 0.000,B 0.000,C 90.000,E1 90.229} C_DIS
LIN {X -0.307,Y -627.923,Z 615.297,A 0.000,B 0.000,C 90.000,E1 89.484} C_DIS
LIN {X 0.120,Y -628.227,Z 615.293,A 0.000,B 0.000,C 90.000,E1 88.682} C_DIS
LIN {X 0.293,Y -628.400,Z 615.287,A 0.000,B 0.000,C 90.000,E1 87.650} C_DIS
LIN {X 0.088,Y -628.310,Z 615.283,A 0.000,B 0.000,C 90.000,E1 86.906} C_DIS
LIN {X 0.303,Y -627.991,Z 615.277,A 0.000,B 0.000,C 90.000,E1 85.869} C_DIS
LIN {X -0.152,Y -627.320,Z 615.272,A 0.000,B 0.000,C 90.000,E1 84.894} C_DIS
LIN {X 0.062,Y -626.523,Z 615.266,A 0.000,B 0.000,C 90.000,E1 83.856} C_DIS
LIN {X -0.131,Y -625.829,Z 615.262,A 0.000,B 0.000,C 90.000,E1 83.109} C_DIS
LIN {X 0.141,Y -624.616,Z 615.256,A 0.000,B 0.000,C 90.000,E1 82.064} C_DIS
LIN {X -0.085,Y -623.490,Z 615.252,A 0.000,B 0.000,C 90.000,E1 81.319} C_DIS
LIN {X -0.291,Y -620.865,Z 615.243,A 0.000,B 0.000,C 90.000,E1 79.803} C_DIS
LIN {X -0.311,Y -618.322,Z 615.236,A 0.000,B 0.000,C 90.000,E1 78.522} C_DIS
LIN {X 0.211,Y -616.675,Z 615.232,A 0.000,B 0.000,C 90.000,E1 77.701} C_DIS
LIN {X -0.120,Y -614.378,Z 615.226,A 0.000,B 0.000,C 90.000,E1 76.700} C_DIS
LIN {X -0.134,Y -611.202,Z 615.219,A 0.000,B 0.000,C 90.000,E1 75.408} C_DIS
LIN {X 0.202,Y -608.517,Z 615.213,A 0.000,B 0.000,C 90.000,E1 74.338} C_DIS
LIN {X -0.083,Y -605.652,Z 615.207,A 0.000,B 0.000,C 90.000,E1 73.323} C_DIS
LIN {X -0.133,Y -603.301,Z 615.203,A 0.000,B 0.000,C 90.000,E1 72.543} C_DIS
LIN {X -0.207,Y -600.728,Z 615.199,A 0.000,B 0.000,C 90.000,E1 71.764} C_DIS
LIN {X 0.154,Y -596.833,Z 615.193,A 0.000,B 0.000,C 90.000,E1 70.678} C_DIS
LIN {X 0.099,Y -592.396,Z 615.187,A 0.000,B 0.000,C 90.000,E1 69.625} C_DIS
LIN {X -0.100,Y -588.908,Z 615.182,A 0.000,B 0.000,C 90.000,E1 68.847} C_DIS
LIN {X 0.090,Y -585.213,Z 615.178,A 0.000,B 0.000,C 90.000,E1 68.028} C_DIS
LIN {X 0.018,Y -581.092,Z 615.174,A 0.000,B 0.000,C 90.000,E1 67.230} C_DIS
LIN {X -0.023,Y -576.719,Z 615.169,A 0.000,B 0.000,C 90.000,E1 66.433} C_DIS
LIN {X 0.200,Y -573.512,Z 615.166,A 0.000,B 0.000,C 90.000,E1 65.869} C_DIS
LIN {X -0.168,Y -569.183,Z 615.162,A 0.000,B 0.000,C 90.000,E1 65.229} C_DIS
LIN {X 0.190,Y -563.440,Z 615.158,A 0.000,B 0.000,C 90.000,E1 64.409} C_DIS
LIN {X 0.189,Y -560.598,Z 615.156,A 0.000,B 0.000,C 90.000,E1 64.024} C_DIS
LIN {X 0.155,Y -556.442,Z 615.153,A 0.000,B 0.000,C 90.000,E1 63.512} C_DIS
LIN {X 0.234,Y -551.843,Z 615.150,A 0.000,B 0.000,C 90.000,E1 62.999} C_DIS
LIN {X -0.090,Y -546.846,Z 615.147,A 0.000,B 0.000,C 90.000,E1 62.538} C_DIS
LIN {X -0.064,Y -541.089,Z 615.145,A 0.000,B 0.000,C 90.000,E1 62.025} C_DIS
LIN {X 0.027,Y -535.000,Z 615.142,A 0.000,B 0.000,C 90.000,E1 61.563} C_DIS
LIN {X -0.221,Y -530.034,Z 615.140,A 0.000,B 0.000,C 90.000,E1 61.257} C_DIS
LIN {X -0.042,Y -523.320,Z 615.138,A 0.000,B 0.000,C 90.000,E1 60.845} C_DIS
LIN {X -0.163,Y -518.498,Z 615.137,A 0.000,B 0.000,C 90.000,E1 60.589} C_DIS
LIN {X 0.149,Y -506.461,Z 615.133,A 0.000,B 0.000,C 90.000,E1 59.950} C_DIS
LIN {X 0.073,Y -482.621,Z 615.127,A 0.000,B 0.000,C 90.000,E1 58.820} C_DIS
LIN {X -0.023,Y -457.428,Z 615.120,A 0.000,B 0.000,C 90.000,E1 57.582} C_DIS
LIN {X 0.082,Y -448.919,Z 615.117,A 0.000,B 0.000,C 90.000,E1 57.120} C_DIS
LIN {X 0.089,Y -444.767,Z 615.116,A 0.000,B 0.000,C 90.000,E1 56.914} C_DIS
LIN {X 0.049,Y -444.696,Z 615.116,A 0.000,B 0.000,C 90.000,E1 56.914} C_DIS
LIN {X -0.016,Y -444.042,Z 615.114,A 0.000,B 0.000,C 90.000,E1 56.548} C_DIS
LIN {X 0.028,Y -434.236,Z 615.090,A 0.000,B 0.000,C 90.000,E1 52.271} C_DIS
LIN {X -0.128,Y -431.748,Z 615.083,A 0.000,B 0.000,C 90.000,E1 50.964} C_DIS
LIN {X 0.051,Y -430.159,Z 615.079,A 0.000,B 0.000,C 90.000,E1 50.275} C_DIS
LIN {X -0.070,Y -428.641,Z 615.076,A 0.000,B 0.000,C 90.000,E1 49.666} C_DIS
LIN {X 0.258,Y -429.507,Z 615.068,A 0.000,B 0.000,C 90.000,E1 48.243} C_DIS
LIN {X -0.173,Y -430.436,Z 615.057,A 0.000,B 0.000,C 90.000,E1 46.296} C_DIS
LIN {X 0.015,Y -431.340,Z 615.046,A 0.000,B 0.000,C 90.000,E1 44.271} C_DIS
LIN {X -0.080,Y -432.374,Z 615.035,A 0.000,B 0.000,C 90.000,E1 42.285} C_DIS
LIN {X -0.128,Y -433.343,Z 615.024,A 0.000,B 0.000,C 90.000,E1 40.297} C_DIS
LIN {X -0.103,Y -434.290,Z 615.013,A 0.000,B 0.000,C 90.000,E1 38.302} C_DIS
LIN {X -0.249,Y -434.974,Z 615.004,A 0.000,B 0.000,C 90.000,E1 36.664} C_DIS
LIN {X -0.022,Y -435.528,Z 614.994,A 0.000,B 0.000,C 90.000,E1 34.978} C_DIS
LIN {X -0.052,Y -435.926,Z 614.987,A 0.000,B 0.000,C 90.000,E1 33.658} C_DIS
LIN {X -0.029,Y -436.406,Z 614.976,A 0.000,B 0.000,C 90.000,E1 31.671} C_DIS
LIN {X 0.140,Y -436.929,Z 614.965,A 0.000,B 0.000,C 90.000,E1 29.667} C_DIS
LIN {X -0.109,Y -437.480,Z 614.954,A 0.000,B 0.000,C 90.000,E1 27.719} C_DIS
LIN {X 0.188,Y -437.858,Z 614.947,A 0.000,B 0.000,C 90.000,E1 26.360} C_DIS
LIN {X -0.013,Y -438.570,Z 614.934,A 0.000,B 0.000,C 90.000,E1 24.079} C_DIS
LIN {X 0.023,Y -439.392,Z 614.921,A 0.000,B 0.000,C 90.000,E1 21.770} C_DIS
LIN {X -0.095,Y -440.257,Z 614.910,A 0.000,B 0.000,C 90.000,E1 19.812} C_DIS
LIN {X 0.053,Y -441.372,Z 614.895,A 0.000,B 0.000,C 90.000,E1 17.166} C_DIS
LIN {X -0.153,Y -442.545,Z 614.883,A 0.000,B 0.000,C 90.000,E1 14.898} C_DIS
LIN {X 0.145,Y -444.099,Z 614.868,A 0.000,B 0.000,C 90.000,E1 12.243} C_DIS
LIN {X -0.141,Y -445.979,Z 614.854,A 0.000,B 0.000,C 90.000,E1 9.670} C_DIS
LIN {X -0.013,Y -447.573,Z 614.843,A 0.000,B 0.000,C 90.000,E1 7.701} C_DIS
LIN {X 0.097,Y -449.359,Z 614.832,A 0.000,B 0.000,C 90.000,E1 5.739} C_DIS
LIN {X -0.090,Y -451.626,Z 614.819,A 0.000,B 0.000,C 90.000,E1 3.498} C_DIS
LIN {X 0.208,Y -454.208,Z 614.807,A 0.000,B 0.000,C 90.000,E1 1.203} C_DIS
LIN {X -0.002,Y -457.738,Z 614.792,A 0.000,B 0.000,C 90.000,E1 358.511} C_DIS
LIN {X 0.208,Y -461.593,Z 614.778,A 0.000,B 0.000,C 90.000,E1 355.931} C_DIS
LIN {X 0.193,Y -465.774,Z 614.763,A 0.000,B 0.000,C 90.000,E1 353.394} C_DIS
LIN {X 0.013,Y -468.414,Z 614.755,A 0.000,B 0.000,C 90.000,E1 351.837} C_DIS
LIN {X -0.060,Y -470.921,Z 614.746,A 0.000,B 0.000,C 90.000,E1 350.274} C_DIS
LIN {X -0.180,Y -474.017,Z 614.736,A 0.000,B 0.000,C 90.000,E1 348.409} C_DIS
LIN {X 0.125,Y -478.381,Z 614.722,A 0.000,B 0.000,C 90.000,E1 345.880} C_DIS
LIN {X 0.050,Y -481.778,Z 614.711,A 0.000,B 0.000,C 90.000,E1 344.031} C_DIS
LIN {X 0.056,Y -485.236,Z 614.701,A 0.000,B 0.000,C 90.000,E1 342.181} C_DIS
LIN {X -0.201,Y -488.213,Z 614.693,A 0.000,B 0.000,C 90.000,E1 340.678} C_DIS
LIN {X -0.075,Y -491.177,Z 614.684,A 0.000,B 0.000,C 90.000,E1 339.135} C_DIS
LIN {X -0.107,Y -493.439,Z 614.677,A 0.000,B 0.000,C 90.000,E1 337.922} C_DIS
LIN {X -0.142,Y -496.063,Z 614.669,A 0.000,B 0.000,C 90.000,E1 336.410} C_DIS
LIN {X -0.116,Y -498.442,Z 614.661,A 0.000,B 0.000,C 90.000,E1 334.897} C_DIS
LIN {X -0.051,Y -500.725,Z 614.652,A 0.000,B 0.000,C 90.000,E1 333.384} C_DIS
LIN {X -0.173,Y -502.942,Z 614.644,A 0.000,B 0.000,C 90.000,E1 331.897} C_DIS
LIN {X -0.012,Y -505.106,Z 614.635,A 0.000,B 0.000,C 90.000,E1 330.383} C_DIS
LIN {X 0.189,Y -507.343,Z 614.627,A 0.000,B 0.000,C 90.000,E1 328.869} C_DIS
LIN {X 0.037,Y -516.486,Z 614.601,A 0.000,B 0.000,C 90.000,E1 324.149} C_DIS
LIN {X 0.088,Y -519.487,Z 614.594,A 0.000,B 0.000,C 90.000,E1 322.970} C_DIS
LIN {X 0.032,Y -520.536,Z 614.593,A 0.000,B 0.000,C 90.000,E1 322.683} C_DIS
LIN {X -0.021,Y -521.439,Z 614.591,A 0.000,B 0.000,C 90.000,E1 322.396} C_DIS
LIN {X -0.072,Y -522.522,Z 614.589,A 0.000,B 0.000,C 90.000,E1 322.110} C_DIS
LIN {X -0.257,Y -523.263,Z 614.589,A 0.000,B 0.000,C 90.000,E1 321.984} C_DIS
LIN {X 0.028,Y -525.696,Z 614.587,A 0.000,B 0.000,C 90.000,E1 321.618} C_DIS
LIN {X -0.010,Y -527.274,Z 614.585,A 0.000,B 0.000,C 90.000,E1 321.331} C_DIS
LIN {X 0.211,Y -536.367,Z 614.580,A 0.000,B 0.000,C 90.000,E1 320.436} C_DIS
LIN {X -0.095,Y -547.271,Z 614.575,A 0.000,B 0.000,C 90.000,E1 319.585} C_DIS
LIN {X 0.085,Y -558.987,Z 614.570,A 0.000,B 0.000,C 90.000,E1 318.647} C_DIS
LIN {X -0.015,Y -574.866,Z 614.563,A 0.000,B 0.000,C 90.000,E1 317.391} C_DIS
LIN {X 0.143,Y -583.535,Z 614.560,A 0.000,B 0.000,C 90.000,E1 316.701} C_DIS
LIN {X -0.163,Y -594.622,Z 614.554,A 0.000,B 0.000,C 90.000,E1 315.810} C_DIS
LIN {X 0.039,Y -602.683,Z 614.551,A 0.000,B 0.000,C 90.000,E1 315.081} C_DIS
LIN {X -0.045,Y -608.986,Z 614.547,A 0.000,B 0.000,C 90.000,E1 314.474} C_DIS
LIN {X -0.171,Y -612.689,Z 614.545,A 0.000,B 0.000,C 90.000,E1 314.109} C_DIS
LIN {X -0.099,Y -618.240,Z 614.542,A 0.000,B 0.000,C 90.000,E1 313.500} C_DIS
LIN {X -0.042,Y -623.868,Z 614.538,A 0.000,B 0.000,C 90.000,E1 312.852} C_DIS
LIN {X -0.071,Y -631.261,Z 614.533,A 0.000,B 0.000,C 90.000,E1 311.962} C_DIS
LIN {X 0.013,Y -639.228,Z 614.528,A 0.000,B 0.000,C 90.000,E1 310.943} C_DIS
LIN {X -0.270,Y -645.937,Z 614.523,A 0.000,B 0.000,C 90.000,E1 310.092} C_DIS
LIN {X 0.081,Y -650.358,Z 614.519,A 0.000,B 0.000,C 90.000,E1 309.439} C_DIS
LIN {X -0.013,Y -653.655,Z 614.516,A 0.000,B 0.000,C 90.000,E1 308.955} C_DIS
LIN {X -0.081,Y -658.146,Z 614.512,A 0.000,B 0.000,C 90.000,E1 308.222} C_DIS
LIN {X -0.069,Y -662.852,Z 614.508,A 0.000,B 0.000,C 90.000,E1 307.363} C_DIS
LIN {X 0.032,Y -665.878,Z 614.504,A 0.000,B 0.000,C 90.000,E1 306.744} C_DIS
LIN {X 0.106,Y -668.181,Z 614.501,A 0.000,B 0.000,C 90.000,E1 306.251} C_DIS
LIN {X 0.168,Y -671.237,Z 614.497,A 0.000,B 0.000,C 90.000,E1 305.518} C_DIS
LIN {X 0.013,Y -674.924,Z 614.492,A 0.000,B 0.000,C 90.000,E1 304.565} C_DIS
LIN {X 0.290,Y -678.371,Z 614.487,A 0.000,B 0.000,C 90.000,E1 303.579} C_DIS
LIN {X 0.234,Y -681.583,Z 614.481,A 0.000,B 0.000,C 90.000,E1 302.625} C_DIS
LIN {X -0.162,Y -685.544,Z 614.475,A 0.000,B 0.000,C 90.000,E1 301.465} C_DIS
LIN {X 0.081,Y -689.342,Z 614.468,A 0.000,B 0.000,C 90.000,E1 300.256} C_DIS
LIN {X 0.038,Y -692.964,Z 614.462,A 0.000,B 0.000,C 90.000,E1 299.077} C_DIS
LIN {X -0.200,Y -695.721,Z 614.456,A 0.000,B 0.000,C 90.000,E1 298.153} C_DIS
LIN {X -0.112,Y -698.254,Z 614.451,A 0.000,B 0.000,C 90.000,E1 297.206} C_DIS
LIN {X 0.062,Y -699.883,Z 614.447,A 0.000,B 0.000,C 90.000,E1 296.488} C_DIS
LIN {X -0.061,Y -700.505,Z 614.443,A 0.000,B 0.000,C 90.000,E1 295.796} C_DIS
LIN {X 0.212,Y -700.157,Z 614.442,A 0.000,B 0.000,C 90.000,E1 295.540} C_DIS
LIN {X 0.122,Y -699.134,Z 614.439,A 0.000,B 0.000,C 90.000,E1 295.079} C_DIS
LIN {X 0.256,Y -698.645,Z 614.439,A 0.000,B 0.000,C 90.000,E1 294.951} C_DIS
LIN {X -0.143,Y -695.252,Z 614.436,A 0.000,B 0.000,C 90.000,E1 294.515} C_DIS
LIN {X -0.015,Y -694.333,Z 614.436,A 0.000,B 0.000,C 90.000,E1 294.387} C_DIS
LIN {X 0.111,Y -692.996,Z 614.435,A 0.000,B 0.000,C 90.000,E1 294.259} C_DIS
LIN {X -0.047,Y -690.832,Z 614.434,A 0.000,B 0.000,C 90.000,E1 294.155} C_DIS
LIN {X 0.146,Y -685.456,Z 614.433,A 0.000,B 0.000,C 90.000,E1 293.898} C_DIS
LIN {X 0.183,Y -683.510,Z 614.432,A 0.000,B 0.000,C 90.000,E1 293.823} C_DIS
LIN {X 0.060,Y -680.942,Z 614.432,A 0.000,B 0.000,C 90.000,E1 293.770} C_DIS
LIN {X -0.027,Y -674.210,Z 614.431,A 0.000,B 0.000,C 90.000,E1 293.643} C_DIS
LIN {X -0.066,Y -657.980,Z 614.430,A 0.000,B 0.000,C 90.000,E1 293.439} C_DIS
LIN {X 0.146,Y -644.013,Z 614.429,A 0.000,B 0.000,C 90.000,E1 293.206} C_DIS
LIN {X 0.083,Y -634.396,Z 614.428,A 0.000,B 0.000,C 90.000,E1 293.025} C_DIS
LIN {X -0.240,Y -624.455,Z 614.427,A 0.000,B 0.000,C 90.000,E1 292.823} C_DIS
LIN {X -0.053,Y -607.846,Z 614.424,A 0.000,B 0.000,C 90.000,E1 292.333} C_DIS
LIN {X -0.203,Y -583.743,Z 614.420,A 0.000,B 0.000,C 90.000,E1 291.589} C_DIS
LIN {X -0.069,Y -576.447,Z 614.419,A 0.000,B 0.000,C 90.000,E1 291.354} C_DIS
LIN {X -0.036,Y -565.946,Z 614.417,A 0.000,B 0.000,C 90.000,E1 291.046} C_DIS
LIN {X 0.205,Y -563.469,Z 614.416,A 0.000,B 0.000,C 90.000,E1 290.918} C_DIS
LIN {X 0.203,Y -559.774,Z 614.415,A 0.000,B 0.000,C 90.000,E1 290.737} C_DIS
LIN {X 0.011,Y -557.852,Z 614.414,A 0.000,B 0.000,C 90.000,E1 290.556} C_DIS
LIN {X -0.031,Y -557.837,Z 614.414,A 0.000,B 0.000,C 90.000,E1 290.556} C_DIS
LIN {X -0.066,Y -557.302,Z 614.413,A 0.000,B 0.000,C 90.000,E1 290.355} C_DIS
LIN {X 0.151,Y -557.085,Z 614.409,A 0.000,B 0.000,C 90.000,E1 289.504} C_DIS
LIN {X -0.095,Y -557.162,Z 614.402,A 0.000,B 0.000,C 90.000,E1 288.417} C_DIS
LIN {X 0.191,Y -557.050,Z 614.396,A 0.000,B 0.000,C 90.000,E1 287.275} C_DIS
LIN {X 0.064,Y -556.605,Z 614.388,A 0.000,B 0.000,C 90.000,E1 285.898} C_DIS
LIN {X 0.186,Y -556.150,Z 614.382,A 0.000,B 0.000,C 90.000,E1 284.773} C_DIS
LIN {X 0.302,Y -555.570,Z 614.376,A 0.000,B 0.000,C 90.000,E1 283.647} C_DIS
LIN {X -0.131,Y -554.856,Z 614.368,A 0.000,B 0.000,C 90.000,E1 282.299} C_DIS
LIN {X -0.032,Y -554.133,Z 614.361,A 0.000,B 0.000,C 90.000,E1 280.894} C_DIS
LIN {X 0.075,Y -553.294,Z 614.351,A 0.000,B 0.000,C 90.000,E1 279.208} C_DIS
LIN {X 0.197,Y -552.359,Z 614.340,A 0.000,B 0.000,C 90.000,E1 277.239} C_DIS
LIN {X 0.118,Y -551.658,Z 614.331,A 0.000,B 0.000,C 90.000,E1 275.568} C_DIS
LIN {X 0.072,Y -551.003,Z 614.320,A 0.000,B 0.000,C 90.000,E1 273.612} C_DIS
LIN {X -0.169,Y -550.571,Z 614.312,A 0.000,B 0.000,C 90.000,E1 272.236} C_DIS
LIN {X 0.133,Y -550.251,Z 614.305,A 0.000,B 0.000,C 90.000,E1 270.802} C_DIS
LIN {X -0.135,Y -549.769,Z 614.297,A 0.000,B 0.000,C 90.000,E1 269.427} C_DIS
LIN {X 0.081,Y -549.321,Z 614.291,A 0.000,B 0.000,C 90.000,E1 268.282} C_DIS
LIN {X -0.118,Y -548.650,Z 614.281,A 0.000,B 0.000,C 90.000,E1 266.617} C_DIS
LIN {X 0.185,Y -547.984,Z 614.273,A 0.000,B 0.000,C 90.000,E1 265.179} C_DIS
LIN {X -0.164,Y -547.283,Z 614.267,A 0.000,B 0.000,C 90.000,E1 264.090} C_DIS
LIN {X 0.045,Y -546.735,Z 614.262,A 0.000,B 0.000,C 90.000,E1 263.223} C_DIS
LIN {X -0.274,Y -545.788,Z 614.256,A 0.000,B 0.000,C 90.000,E1 262.129} C_DIS
LIN {X 0.182,Y -544.113,Z 614.247,A 0.000,B 0.000,C 90.000,E1 260.387} C_DIS
LIN {X -0.224,Y -541.657,Z 614.233,A 0.000,B 0.000,C 90.000,E1 257.881} C_DIS
LIN {X -0.172,Y -540.137,Z 614.223,A 0.000,B 0.000,C 90.000,E1 256.172} C_DIS
LIN {X -0.218,Y -538.786,Z 614.215,A 0.000,B 0.000,C 90.000,E1 254.755} C_DIS
LIN {X 0.057,Y -536.925,Z 614.206,A 0.000,B 0.000,C 90.000,E1 253.015} C_DIS
LIN {X -0.210,Y -535.234,Z 614.196,A 0.000,B 0.000,C 90.000,E1 251.329} C_DIS
LIN {X -0.247,Y -533.893,Z 614.190,A 0.000,B 0.000,C 90.000,E1 250.188} C_DIS
LIN {X -0.141,Y -532.670,Z 614.185,A 0.000,B 0.000,C 90.000,E1 249.316} C_DIS
LIN {X 0.156,Y -530.380,Z 614.177,A 0.000,B 0.000,C 90.000,E1 247.847} C_DIS
LIN {X -0.276,Y -528.349,Z 614.171,A 0.000,B 0.000,C 90.000,E1 246.741} C_DIS
LIN {X 0.166,Y -526.225,Z 614.164,A 0.000,B 0.000,C 90.000,E1 245.537} C_DIS
LIN {X -0.119,Y -523.822,Z 614.158,A 0.000,B 0.000,C 90.000,E1 244.409} C_DIS
LIN {X -0.214,Y -521.309,Z 614.151,A 0.000,B 0.000,C 90.000,E1 243.256} C_DIS
LIN {X -0.102,Y -518.726,Z 614.145,A 0.000,B 0.000,C 90.000,E1 242.076} C_DIS
LIN {X 0.091,Y -515.343,Z 614.137,A 0.000,B 0.000,C 90.000,E1 240.589} C_DIS
LIN {X 0.102,Y -511.193,Z 614.127,A 0.000,B 0.000,C 90.000,E1 238.820} C_DIS
LIN {X -0.116,Y -508.239,Z 614.120,A 0.000,B 0.000,C 90.000,E1 237.661} C_DIS
LIN {X -0.058,Y -504.346,Z 614.112,A 0.000,B 0.000,C 90.000,E1 236.167} C_DIS
LIN {X -0.208,Y -500.276,Z 614.104,A 0.000,B 0.000,C 90.000,E1 234.689} C_DIS
LIN {X -0.004,Y -494.660,Z 614.092,A 0.000,B 0.000,C 90.000,E1 232.557} C_DIS
LIN {X -0.037,Y -490.885,Z 614.084,A 0.000,B 0.000,C 90.000,E1 231.045} C_DIS
LIN {X -0.100,Y -484.658,Z 614.070,A 0.000,B 0.000,C 90.000,E1 228.609} C_DIS
LIN {X 0.062,Y -480.072,Z 614.060,A 0.000,B 0.000,C 90.000,E1 226.743} C_DIS
LIN {X -0.017,Y -474.034,Z 614.046,A 0.000,B 0.000,C 90.000,E1 224.271} C_DIS
LIN {X -0.015,Y -469.046,Z 614.034,A 0.000,B 0.000,C 90.000,E1 222.081} C_DIS
LIN {X -0.274,Y -465.550,Z 614.025,A 0.000,B 0.000,C 90.000,E1 220.539} C_DIS
LIN {X -0.145,Y -461.470,Z 614.015,A 0.000,B 0.000,C 90.000,E1 218.624} C_DIS
LIN {X -0.115,Y -457.565,Z 614.004,A 0.000,B 0.000,C 90.000,E1 216.710} C_DIS
LIN {X -0.007,Y -453.236,Z 613.991,A 0.000,B 0.000,C 90.000,E1 214.452} C_DIS
LIN {X 0.067,Y -450.266,Z 613.982,A 0.000,B 0.000,C 90.000,E1 212.832} C_DIS
LIN {X -0.145,Y -446.143,Z 613.970,A 0.000,B 0.000,C 90.000,E1 210.590} C_DIS
LIN {X 0.008,Y -442.723,Z 613.959,A 0.000,B 0.000,C 90.000,E1 208.615} C_DIS
LIN {X -0.172,Y -439.775,Z 613.950,A 0.000,B 0.000,C 90.000,E1 207.001} C_DIS
LIN {X -0.039,Y -437.473,Z 613.943,A 0.000,B 0.000,C 90.000,E1 205.668} C_DIS
LIN {X 0.114,Y -433.462,Z 613.930,A 0.000,B 0.000,C 90.000,E1 203.334} C_DIS
LIN {X -0.187,Y -429.561,Z 613.917,A 0.000,B 0.000,C 90.000,E1 201.046} C_DIS
LIN {X -0.142,Y -426.225,Z 613.906,A 0.000,B 0.000,C 90.000,E1 199.033} C_DIS
LIN {X 0.087,Y -423.111,Z 613.894,A 0.000,B 0.000,C 90.000,E1 196.985} C_DIS
LIN {X -0.125,Y -419.745,Z 613.881,A 0.000,B 0.000,C 90.000,E1 194.647} C_DIS
LIN {X -0.197,Y -417.735,Z 613.874,A 0.000,B 0.000,C 90.000,E1 193.300} C_DIS
LIN {X -0.017,Y -413.619,Z 613.859,A 0.000,B 0.000,C 90.000,E1 190.546} C_DIS
LIN {X -0.187,Y -410.840,Z 613.847,A 0.000,B 0.000,C 90.000,E1 188.511} C_DIS
LIN {X -0.102,Y -408.532,Z 613.838,A 0.000,B 0.000,C 90.000,E1 186.777} C_DIS
LIN {X -0.105,Y -405.898,Z 613.826,A 0.000,B 0.000,C 90.000,E1 184.702} C_DIS
LIN {X 0.001,Y -401.717,Z 613.805,A 0.000,B 0.000,C 90.000,E1 180.859} C_DIS
LIN {X -0.116,Y -398.551,Z 613.781,A 0.000,B 0.000,C 90.000,E1 176.674} C_DIS
LIN {X 0.193,Y -397.041,Z 613.760,A 0.000,B 0.000,C 90.000,E1 172.761} C_DIS
LIN {X -0.076,Y -396.549,Z 613.744,A 0.000,B 0.000,C 90.000,E1 169.982} C_DIS
LIN {X -0.150,Y -396.522,Z 613.729,A 0.000,B 0.000,C 90.000,E1 167.173} C_DIS
LIN {X -0.040,Y -396.993,Z 613.713,A 0.000,B 0.000,C 90.000,E1 164.338} C_DIS
LIN {X 0.195,Y -397.383,Z 613.703,A 0.000,B 0.000,C 90.000,E1 162.543} C_DIS
LIN {X -0.044,Y -397.994,Z 613.690,A 0.000,B 0.000,C 90.000,E1 160.115} C_DIS
LIN {X 0.098,Y -398.586,Z 613.680,A 0.000,B 0.000,C 90.000,E1 158.337} C_DIS
LIN {X -0.127,Y -399.188,Z 613.670,A 0.000,B 0.000,C 90.000,E1 156.613} C_DIS
LIN {X -0.087,Y -400.121,Z 613.656,A 0.000,B 0.000,C 90.000,E1 154.152} C_DIS
LIN {X -0.031,Y -400.622,Z 613.649,A 0.000,B 0.000,C 90.000,E1 152.743} C_DIS
LIN {X 0.220,Y -401.145,Z 613.641,A 0.000,B 0.000,C 90.000,E1 151.307} C_DIS
LIN {X -0.083,Y -401.818,Z 613.629,A 0.000,B 0.000,C 90.000,E1 149.253} C_DIS
LIN {X -0.059,Y -402.313,Z 613.619,A 0.000,B 0.000,C 90.000,E1 147.502} C_DIS
